gfCNCPoint2[20411] = {X 393.9120, Y 101.1273, Z -3.0000, A 0.000, B 0.000, C 0.000 }
gfCNCPoint2[20412] = {X 393.2786, Y 100.4940, Z -3.0000, A 0.000, B 0.000, C 0.000 }
gfCNCPoint2[20413] = {X 392.8021, Y 99.7355, Z -3.0000, A 0.000, B 0.000, C 0.000 }
gfCNCPoint2[20414] = {X 392.5062, Y 98.8901, Z -3.0000, A 0.000, B 0.000, C 0.000 }
gfCNCPoint2[20415] = {X 392.4059, Y 98.0000, Z -3.0000, A 0.000, B 0.000, C 0.000 }
gfCNCPoint2[20416] = {X 392.4059, Y 97.0659, Z -3.0000, A 0.000, B 0.000, C 0.000 }
gfCNCPoint2[20417] = {X 392.5058, Y 96.1776, Z -3.0000, A 0.000, B 0.000, C 0.000 }
gfCNCPoint2[20418] = {X 392.8005, Y 95.3337, Z -3.0000, A 0.000, B 0.000, C 0.000 }
gfCNCPoint2[20419] = {X 393.2753, Y 94.5762, Z -3.0000, A 0.000, B 0.000, C 0.000 }
gfCNCPoint2[20420] = {X 393.9064, Y 93.9431, Z -3.0000, A 0.000, B 0.000, C 0.000 }
gfCNCPoint2[20421] = {X 394.6623, Y 93.4660, Z -3.0000, A 0.000, B 0.000, C 0.000 }
gfCNCPoint2[20422] = {X 395.5053, Y 93.1686, Z -3.0000, A 0.000, B 0.000, C 0.000 }
gfCNCPoint2[20423] = {X 396.3933, Y 93.0660, Z -3.0000, A 0.000, B 0.000, C 0.000 }
gfCNCPoint2[20424] = {X 397.3648, Y 93.0246, Z -3.0000, A 0.000, B 0.000, C 0.000 }
gfCNCPoint2[20425] = {X 398.3327, Y 92.9326, Z -3.0000, A 0.000, B 0.000, C 0.000 }
gfCNCPoint2[20426] = {X 399.0538, Y 92.7580, Z -3.0000, A 0.000, B 0.000, C 0.000 }
gfCNCPoint2[20427] = {X 399.7177, Y 92.4268, Z -3.0000, A 0.000, B 0.000, C 0.000 }
gfCNCPoint2[20428] = {X 405.3929, Y 88.7698, Z -3.0000, A 0.000, B 0.000, C 0.000 }
gfCNCPoint2[20429] = {X 413.9654, Y 83.2883, Z -3.0000, A 0.000, B 0.000, C 0.000 }
gfCNCPoint2[20430] = {X 411.7675, Y 79.8509, Z -3.0000, A 0.000, B 0.000, C 0.000 }
gfCNCPoint2[20431] = {X 411.7675, Y 79.8509, Z 0.0000, A 0.000, B 0.000, C 0.000 }
gfCNCPoint2[20432] = {X 411.7675, Y 79.8509, Z 11.0000, A 0.000, B 0.000, C 0.000 }
gfCNCPoint2[20433] = {X 466.3102, Y 28.5935, Z 11.0000, A 0.000, B 0.000, C 0.000 }
gfCNCPoint2[20434] = {X 466.3102, Y 28.5935, Z 0.0000, A 0.000, B 0.000, C 0.000 }
gfCNCPoint2[20435] = {X 466.3102, Y 28.5935, Z -3.0000, A 0.000, B 0.000, C 0.000 }
gfCNCPoint2[20436] = {X 462.2302, Y 28.5935, Z -3.0000, A 0.000, B 0.000, C 0.000 }
gfCNCPoint2[20437] = {X 462.2304, Y 40.9130, Z -3.0000, A 0.000, B 0.000, C 0.000 }
gfCNCPoint2[20438] = {X 462.2392, Y 40.9201, Z -3.0000, A 0.000, B 0.000, C 0.000 }
gfCNCPoint2[20439] = {X 462.8741, Y 41.5906, Z -3.0000, A 0.000, B 0.000, C 0.000 }
gfCNCPoint2[20440] = {X 463.3521, Y 42.3808, Z -3.0000, A 0.000, B 0.000, C 0.000 }
gfCNCPoint2[20441] = {X 463.6512, Y 43.2545, Z -3.0000, A 0.000, B 0.000, C 0.000 }
gfCNCPoint2[20442] = {X 463.7578, Y 44.1718, Z -3.0000, A 0.000, B 0.000, C 0.000 }
gfCNCPoint2[20443] = {X 463.7579, Y 45.0000, Z -3.0000, A 0.000, B 0.000, C 0.000 }
gfCNCPoint2[20444] = {X 463.6496, Y 45.9613, Z -3.0000, A 0.000, B 0.000, C 0.000 }
gfCNCPoint2[20445] = {X 463.3301, Y 46.8744, Z -3.0000, A 0.000, B 0.000, C 0.000 }
gfCNCPoint2[20446] = {X 462.8155, Y 47.6935, Z -3.0000, A 0.000, B 0.000, C 0.000 }
gfCNCPoint2[20447] = {X 462.1314, Y 48.3775, Z -3.0000, A 0.000, B 0.000, C 0.000 }
gfCNCPoint2[20448] = {X 461.3123, Y 48.8922, Z -3.0000, A 0.000, B 0.000, C 0.000 }
gfCNCPoint2[20449] = {X 460.3992, Y 49.2117, Z -3.0000, A 0.000, B 0.000, C 0.000 }
gfCNCPoint2[20450] = {X 459.4379, Y 49.3200, Z -3.0000, A 0.000, B 0.000, C 0.000 }
gfCNCPoint2[20451] = {X 452.9945, Y 49.3200, Z -3.0000, A 0.000, B 0.000, C 0.000 }
gfCNCPoint2[20452] = {X 452.0381, Y 49.2128, Z -3.0000, A 0.000, B 0.000, C 0.000 }
gfCNCPoint2[20453] = {X 451.1291, Y 48.8965, Z -3.0000, A 0.000, B 0.000, C 0.000 }
gfCNCPoint2[20454] = {X 450.3127, Y 48.3868, Z -3.0000, A 0.000, B 0.000, C 0.000 }
gfCNCPoint2[20455] = {X 449.6294, Y 47.7091, Z -3.0000, A 0.000, B 0.000, C 0.000 }
gfCNCPoint2[20456] = {X 449.1132, Y 46.8968, Z -3.0000, A 0.000, B 0.000, C 0.000 }
gfCNCPoint2[20457] = {X 448.7895, Y 45.9905, Z -3.0000, A 0.000, B 0.000, C 0.000 }
gfCNCPoint2[20458] = {X 448.6746, Y 45.0349, Z -3.0000, A 0.000, B 0.000, C 0.000 }
gfCNCPoint2[20459] = {X 448.6749, Y 44.1494, Z -3.0000, A 0.000, B 0.000, C 0.000 }
gfCNCPoint2[20460] = {X 448.7853, Y 43.2364, Z -3.0000, A 0.000, B 0.000, C 0.000 }
gfCNCPoint2[20461] = {X 449.0865, Y 42.3675, Z -3.0000, A 0.000, B 0.000, C 0.000 }
gfCNCPoint2[20462] = {X 449.5648, Y 41.5821, Z -3.0000, A 0.000, B 0.000, C 0.000 }
gfCNCPoint2[20463] = {X 450.1984, Y 40.9157, Z -3.0000, A 0.000, B 0.000, C 0.000 }
gfCNCPoint2[20464] = {X 450.1984, Y 34.4738, Z -3.0000, A 0.000, B 0.000, C 0.000 }
gfCNCPoint2[20465] = {X 447.4740, Y 34.4738, Z -3.0000, A 0.000, B 0.000, C 0.000 }
gfCNCPoint2[20466] = {X 443.1893, Y 42.8160, Z -3.0000, A 0.000, B 0.000, C 0.000 }
gfCNCPoint2[20467] = {X 443.1944, Y 42.8296, Z -3.0000, A 0.000, B 0.000, C 0.000 }
gfCNCPoint2[20468] = {X 443.3604, Y 43.4910, Z -3.0000, A 0.000, B 0.000, C 0.000 }
gfCNCPoint2[20469] = {X 443.4203, Y 44.1703, Z -3.0000, A 0.000, B 0.000, C 0.000 }
gfCNCPoint2[20470] = {X 443.4205, Y 45.0000, Z -3.0000, A 0.000, B 0.000, C 0.000 }
gfCNCPoint2[20471] = {X 443.3122, Y 45.9613, Z -3.0000, A 0.000, B 0.000, C 0.000 }
gfCNCPoint2[20472] = {X 442.9927, Y 46.8744, Z -3.0000, A 0.000, B 0.000, C 0.000 }
gfCNCPoint2[20473] = {X 442.4780, Y 47.6935, Z -3.0000, A 0.000, B 0.000, C 0.000 }
gfCNCPoint2[20474] = {X 441.7939, Y 48.3775, Z -3.0000, A 0.000, B 0.000, C 0.000 }
gfCNCPoint2[20475] = {X 440.9748, Y 48.8922, Z -3.0000, A 0.000, B 0.000, C 0.000 }
gfCNCPoint2[20476] = {X 440.0618, Y 49.2117, Z -3.0000, A 0.000, B 0.000, C 0.000 }
gfCNCPoint2[20477] = {X 439.1005, Y 49.3200, Z -3.0000, A 0.000, B 0.000, C 0.000 }
gfCNCPoint2[20478] = {X 432.5144, Y 49.3200, Z -3.0000, A 0.000, B 0.000, C 0.000 }
gfCNCPoint2[20479] = {X 431.5531, Y 49.2117, Z -3.0000, A 0.000, B 0.000, C 0.000 }
gfCNCPoint2[20480] = {X 430.6401, Y 48.8922, Z -3.0000, A 0.000, B 0.000, C 0.000 }
gfCNCPoint2[20481] = {X 429.8210, Y 48.3775, Z -3.0000, A 0.000, B 0.000, C 0.000 }
gfCNCPoint2[20482] = {X 429.1369, Y 47.6935, Z -3.0000, A 0.000, B 0.000, C 0.000 }
gfCNCPoint2[20483] = {X 428.6223, Y 46.8745, Z -3.0000, A 0.000, B 0.000, C 0.000 }
gfCNCPoint2[20484] = {X 428.3027, Y 45.9614, Z -3.0000, A 0.000, B 0.000, C 0.000 }
gfCNCPoint2[20485] = {X 428.1944, Y 45.0001, Z -3.0000, A 0.000, B 0.000, C 0.000 }
gfCNCPoint2[20486] = {X 428.1948, Y 44.1494, Z -3.0000, A 0.000, B 0.000, C 0.000 }
gfCNCPoint2[20487] = {X 428.2925, Y 43.2935, Z -3.0000, A 0.000, B 0.000, C 0.000 }
gfCNCPoint2[20488] = {X 428.5580, Y 42.4740, Z -3.0000, A 0.000, B 0.000, C 0.000 }
gfCNCPoint2[20489] = {X 428.9809, Y 41.7236, Z -3.0000, A 0.000, B 0.000, C 0.000 }
gfCNCPoint2[20490] = {X 429.5442, Y 41.0719, Z -3.0000, A 0.000, B 0.000, C 0.000 }
gfCNCPoint2[20491] = {X 430.2256, Y 40.5449, Z -3.0000, A 0.000, B 0.000, C 0.000 }
gfCNCPoint2[20492] = {X 430.9981, Y 40.1637, Z -3.0000, A 0.000, B 0.000, C 0.000 }
gfCNCPoint2[20493] = {X 434.9873, Y 32.3552, Z -3.0000, A 0.000, B 0.000, C 0.000 }
gfCNCPoint2[20494] = {X 433.8174, Y 31.5687, Z -3.0000, A 0.000, B 0.000, C 0.000 }
gfCNCPoint2[20495] = {X 432.7544, Y 30.6429, Z -3.0000, A 0.000, B 0.000, C 0.000 }
gfCNCPoint2[20496] = {X 431.8146, Y 29.5922, Z -3.0000, A 0.000, B 0.000, C 0.000 }
gfCNCPoint2[20497] = {X 431.0127, Y 28.4328, Z -3.0000, A 0.000, B 0.000, C 0.000 }
gfCNCPoint2[20498] = {X 430.3611, Y 27.1828, Z -3.0000, A 0.000, B 0.000, C 0.000 }
gfCNCPoint2[20499] = {X 429.8699, Y 25.8615, Z -3.0000, A 0.000, B 0.000, C 0.000 }
gfCNCPoint2[20500] = {X 429.4508, Y 24.0500, Z -3.0000, A 0.000, B 0.000, C 0.000 }
gfCNCPoint2[20501] = {X 429.2372, Y 22.2029, Z -3.0000, A 0.000, B 0.000, C 0.000 }
gfCNCPoint2[20502] = {X 429.2318, Y 20.3436, Z -3.0000, A 0.000, B 0.000, C 0.000 }
gfCNCPoint2[20503] = {X 429.4347, Y 18.4953, Z -3.0000, A 0.000, B 0.000, C 0.000 }
gfCNCPoint2[20504] = {X 429.8434, Y 16.6814, Z -3.0000, A 0.000, B 0.000, C 0.000 }
gfCNCPoint2[20505] = {X 430.3648, Y 15.2116, Z -3.0000, A 0.000, B 0.000, C 0.000 }
gfCNCPoint2[20506] = {X 431.0757, Y 13.8235, Z -3.0000, A 0.000, B 0.000, C 0.000 }
gfCNCPoint2[20507] = {X 431.9635, Y 12.5413, Z -3.0000, A 0.000, B 0.000, C 0.000 }
gfCNCPoint2[20508] = {X 433.0127, Y 11.3874, Z -3.0000, A 0.000, B 0.000, C 0.000 }
gfCNCPoint2[20509] = {X 434.2050, Y 10.3821, Z -3.0000, A 0.000, B 0.000, C 0.000 }
gfCNCPoint2[20510] = {X 435.5195, Y 9.5429, Z -3.0000, A 0.000, B 0.000, C 0.000 }
gfCNCPoint2[20511] = {X 436.9333, Y 8.8845, Z -3.0000, A 0.000, B 0.000, C 0.000 }
gfCNCPoint2[20512] = {X 438.4216, Y 8.4184, Z -3.0000, A 0.000, B 0.000, C 0.000 }
gfCNCPoint2[20513] = {X 440.0467, Y 8.1096, Z -3.0000, A 0.000, B 0.000, C 0.000 }
gfCNCPoint2[20514] = {X 441.6910, Y 7.9282, Z -3.0000, A 0.000, B 0.000, C 0.000 }
gfCNCPoint2[20515] = {X 443.3444, Y 7.8753, Z -3.0000, A 0.000, B 0.000, C 0.000 }
gfCNCPoint2[20516] = {X 444.0357, Y 7.8712, Z -3.0000, A 0.000, B 0.000, C 0.000 }
gfCNCPoint2[20517] = {X 459.4466, Y 7.8712, Z -3.0000, A 0.000, B 0.000, C 0.000 }
gfCNCPoint2[20518] = {X 460.4060, Y 7.9793, Z -3.0000, A 0.000, B 0.000, C 0.000 }
gfCNCPoint2[20519] = {X 461.3172, Y 8.2982, Z -3.0000, A 0.000, B 0.000, C 0.000 }
gfCNCPoint2[20520] = {X 462.1347, Y 8.8118, Z -3.0000, A 0.000, B 0.000, C 0.000 }
gfCNCPoint2[20521] = {X 462.8173, Y 9.4945, Z -3.0000, A 0.000, B 0.000, C 0.000 }
gfCNCPoint2[20522] = {X 463.3310, Y 10.3120, Z -3.0000, A 0.000, B 0.000, C 0.000 }
gfCNCPoint2[20523] = {X 463.6498, Y 11.2232, Z -3.0000, A 0.000, B 0.000, C 0.000 }
gfCNCPoint2[20524] = {X 463.7579, Y 12.1826, Z -3.0000, A 0.000, B 0.000, C 0.000 }
gfCNCPoint2[20525] = {X 463.7579, Y 12.9781, Z -3.0000, A 0.000, B 0.000, C 0.000 }
gfCNCPoint2[20526] = {X 463.6565, Y 13.9081, Z -3.0000, A 0.000, B 0.000, C 0.000 }
gfCNCPoint2[20527] = {X 463.3573, Y 14.7945, Z -3.0000, A 0.000, B 0.000, C 0.000 }
gfCNCPoint2[20528] = {X 462.8742, Y 15.5957, Z -3.0000, A 0.000, B 0.000, C 0.000 }
gfCNCPoint2[20529] = {X 462.2300, Y 16.2741, Z -3.0000, A 0.000, B 0.000, C 0.000 }
gfCNCPoint2[20530] = {X 462.2302, Y 28.5935, Z -3.0000, A 0.000, B 0.000, C 0.000 }
gfCNCPoint2[20531] = {X 466.2302, Y 28.5935, Z -3.0000, A 0.000, B 0.000, C 0.000 }
gfCNCPoint2[20532] = {X 462.1502, Y 28.5935, Z -3.0000, A 0.000, B 0.000, C 0.000 }
gfCNCPoint2[20533] = {X 462.1504, Y 40.9512, Z -3.0000, A 0.000, B 0.000, C 0.000 }
gfCNCPoint2[20534] = {X 462.1880, Y 40.9816, Z -3.0000, A 0.000, B 0.000, C 0.000 }
gfCNCPoint2[20535] = {X 462.8110, Y 41.6397, Z -3.0000, A 0.000, B 0.000, C 0.000 }
gfCNCPoint2[20536] = {X 463.2798, Y 42.4151, Z -3.0000, A 0.000, B 0.000, C 0.000 }
gfCNCPoint2[20537] = {X 463.5732, Y 43.2724, Z -3.0000, A 0.000, B 0.000, C 0.000 }
gfCNCPoint2[20538] = {X 463.6778, Y 44.1724, Z -3.0000, A 0.000, B 0.000, C 0.000 }
gfCNCPoint2[20539] = {X 463.6779, Y 45.0000, Z -3.0000, A 0.000, B 0.000, C 0.000 }
gfCNCPoint2[20540] = {X 463.5716, Y 45.9435, Z -3.0000, A 0.000, B 0.000, C 0.000 }
gfCNCPoint2[20541] = {X 463.2580, Y 46.8397, Z -3.0000, A 0.000, B 0.000, C 0.000 }
gfCNCPoint2[20542] = {X 462.7529, Y 47.6436, Z -3.0000, A 0.000, B 0.000, C 0.000 }
gfCNCPoint2[20543] = {X 462.0815, Y 48.3150, Z -3.0000, A 0.000, B 0.000, C 0.000 }
gfCNCPoint2[20544] = {X 461.2776, Y 48.8201, Z -3.0000, A 0.000, B 0.000, C 0.000 }
gfCNCPoint2[20545] = {X 460.3814, Y 49.1337, Z -3.0000, A 0.000, B 0.000, C 0.000 }
gfCNCPoint2[20546] = {X 459.4379, Y 49.2400, Z -3.0000, A 0.000, B 0.000, C 0.000 }
gfCNCPoint2[20547] = {X 452.9945, Y 49.2400, Z -3.0000, A 0.000, B 0.000, C 0.000 }
gfCNCPoint2[20548] = {X 452.0558, Y 49.1348, Z -3.0000, A 0.000, B 0.000, C 0.000 }
gfCNCPoint2[20549] = {X 451.1636, Y 48.8243, Z -3.0000, A 0.000, B 0.000, C 0.000 }
gfCNCPoint2[20550] = {X 450.3624, Y 48.3241, Z -3.0000, A 0.000, B 0.000, C 0.000 }
gfCNCPoint2[20551] = {X 449.6918, Y 47.6589, Z -3.0000, A 0.000, B 0.000, C 0.000 }
gfCNCPoint2[20552] = {X 449.1851, Y 46.8617, Z -3.0000, A 0.000, B 0.000, C 0.000 }
gfCNCPoint2[20553] = {X 448.8674, Y 45.9721, Z -3.0000, A 0.000, B 0.000, C 0.000 }
gfCNCPoint2[20554] = {X 448.7546, Y 45.0343, Z -3.0000, A 0.000, B 0.000, C 0.000 }
gfCNCPoint2[20555] = {X 448.7549, Y 44.1505, Z -3.0000, A 0.000, B 0.000, C 0.000 }
gfCNCPoint2[20556] = {X 448.8654, Y 43.2454, Z -3.0000, A 0.000, B 0.000, C 0.000 }
gfCNCPoint2[20557] = {X 449.1668, Y 42.3850, Z -3.0000, A 0.000, B 0.000, C 0.000 }
gfCNCPoint2[20558] = {X 449.6452, Y 41.6088, Z -3.0000, A 0.000, B 0.000, C 0.000 }
gfCNCPoint2[20559] = {X 450.2784, Y 40.9529, Z -3.0000, A 0.000, B 0.000, C 0.000 }
gfCNCPoint2[20560] = {X 450.2784, Y 34.3938, Z -3.0000, A 0.000, B 0.000, C 0.000 }
gfCNCPoint2[20561] = {X 447.4251, Y 34.3938, Z -3.0000, A 0.000, B 0.000, C 0.000 }
gfCNCPoint2[20562] = {X 443.1021, Y 42.8107, Z -3.0000, A 0.000, B 0.000, C 0.000 }
gfCNCPoint2[20563] = {X 443.1190, Y 42.8563, Z -3.0000, A 0.000, B 0.000, C 0.000 }
gfCNCPoint2[20564] = {X 443.2816, Y 43.5049, Z -3.0000, A 0.000, B 0.000, C 0.000 }
gfCNCPoint2[20565] = {X 443.3403, Y 44.1710, Z -3.0000, A 0.000, B 0.000, C 0.000 }
gfCNCPoint2[20566] = {X 443.3405, Y 45.0000, Z -3.0000, A 0.000, B 0.000, C 0.000 }
gfCNCPoint2[20567] = {X 443.2342, Y 45.9435, Z -3.0000, A 0.000, B 0.000, C 0.000 }
gfCNCPoint2[20568] = {X 442.9206, Y 46.8397, Z -3.0000, A 0.000, B 0.000, C 0.000 }
gfCNCPoint2[20569] = {X 442.4154, Y 47.6436, Z -3.0000, A 0.000, B 0.000, C 0.000 }
gfCNCPoint2[20570] = {X 441.7441, Y 48.3150, Z -3.0000, A 0.000, B 0.000, C 0.000 }
gfCNCPoint2[20571] = {X 440.9401, Y 48.8201, Z -3.0000, A 0.000, B 0.000, C 0.000 }
gfCNCPoint2[20572] = {X 440.0440, Y 49.1337, Z -3.0000, A 0.000, B 0.000, C 0.000 }
gfCNCPoint2[20573] = {X 439.1005, Y 49.2400, Z -3.0000, A 0.000, B 0.000, C 0.000 }
gfCNCPoint2[20574] = {X 432.5144, Y 49.2400, Z -3.0000, A 0.000, B 0.000, C 0.000 }
gfCNCPoint2[20575] = {X 431.5709, Y 49.1337, Z -3.0000, A 0.000, B 0.000, C 0.000 }
gfCNCPoint2[20576] = {X 430.6748, Y 48.8201, Z -3.0000, A 0.000, B 0.000, C 0.000 }
gfCNCPoint2[20577] = {X 429.8708, Y 48.3150, Z -3.0000, A 0.000, B 0.000, C 0.000 }
gfCNCPoint2[20578] = {X 429.1995, Y 47.6436, Z -3.0000, A 0.000, B 0.000, C 0.000 }
gfCNCPoint2[20579] = {X 428.6943, Y 46.8397, Z -3.0000, A 0.000, B 0.000, C 0.000 }
gfCNCPoint2[20580] = {X 428.3807, Y 45.9436, Z -3.0000, A 0.000, B 0.000, C 0.000 }
gfCNCPoint2[20581] = {X 428.2744, Y 45.0001, Z -3.0000, A 0.000, B 0.000, C 0.000 }
gfCNCPoint2[20582] = {X 428.2748, Y 44.1505, Z -3.0000, A 0.000, B 0.000, C 0.000 }
gfCNCPoint2[20583] = {X 428.3718, Y 43.3054, Z -3.0000, A 0.000, B 0.000, C 0.000 }
gfCNCPoint2[20584] = {X 428.6354, Y 42.4967, Z -3.0000, A 0.000, B 0.000, C 0.000 }
gfCNCPoint2[20585] = {X 429.0552, Y 41.7570, Z -3.0000, A 0.000, B 0.000, C 0.000 }
gfCNCPoint2[20586] = {X 429.6142, Y 41.1159, Z -3.0000, A 0.000, B 0.000, C 0.000 }
gfCNCPoint2[20587] = {X 430.2899, Y 40.5992, Z -3.0000, A 0.000, B 0.000, C 0.000 }
gfCNCPoint2[20588] = {X 431.0551, Y 40.2278, Z -3.0000, A 0.000, B 0.000, C 0.000 }
gfCNCPoint2[20589] = {X 435.0930, Y 32.3241, Z -3.0000, A 0.000, B 0.000, C 0.000 }
gfCNCPoint2[20590] = {X 433.9162, Y 31.5434, Z -3.0000, A 0.000, B 0.000, C 0.000 }
gfCNCPoint2[20591] = {X 432.8465, Y 30.6212, Z -3.0000, A 0.000, B 0.000, C 0.000 }
gfCNCPoint2[20592] = {X 431.9009, Y 29.5723, Z -3.0000, A 0.000, B 0.000, C 0.000 }
gfCNCPoint2[20593] = {X 431.0943, Y 28.4130, Z -3.0000, A 0.000, B 0.000, C 0.000 }
gfCNCPoint2[20594] = {X 430.4394, Y 27.1618, Z -3.0000, A 0.000, B 0.000, C 0.000 }
gfCNCPoint2[20595] = {X 429.9465, Y 25.8383, Z -3.0000, A 0.000, B 0.000, C 0.000 }
gfCNCPoint2[20596] = {X 429.5295, Y 24.0357, Z -3.0000, A 0.000, B 0.000, C 0.000 }
gfCNCPoint2[20597] = {X 429.3171, Y 22.1977, Z -3.0000, A 0.000, B 0.000, C 0.000 }
gfCNCPoint2[20598] = {X 429.3117, Y 20.3474, Z -3.0000, A 0.000, B 0.000, C 0.000 }
gfCNCPoint2[20599] = {X 429.5137, Y 18.5082, Z -3.0000, A 0.000, B 0.000, C 0.000 }
gfCNCPoint2[20600] = {X 429.9203, Y 16.7032, Z -3.0000, A 0.000, B 0.000, C 0.000 }
gfCNCPoint2[20601] = {X 430.4383, Y 15.2434, Z -3.0000, A 0.000, B 0.000, C 0.000 }
gfCNCPoint2[20602] = {X 431.1443, Y 13.8646, Z -3.0000, A 0.000, B 0.000, C 0.000 }
gfCNCPoint2[20603] = {X 432.0261, Y 12.5911, Z -3.0000, A 0.000, B 0.000, C 0.000 }
gfCNCPoint2[20604] = {X 433.0682, Y 11.4451, Z -3.0000, A 0.000, B 0.000, C 0.000 }
gfCNCPoint2[20605] = {X 434.2524, Y 10.4466, Z -3.0000, A 0.000, B 0.000, C 0.000 }
gfCNCPoint2[20606] = {X 435.5580, Y 9.6131, Z -3.0000, A 0.000, B 0.000, C 0.000 }
gfCNCPoint2[20607] = {X 436.9622, Y 8.9591, Z -3.0000, A 0.000, B 0.000, C 0.000 }
gfCNCPoint2[20608] = {X 438.4404, Y 8.4961, Z -3.0000, A 0.000, B 0.000, C 0.000 }
gfCNCPoint2[20609] = {X 440.0593, Y 8.1886, Z -3.0000, A 0.000, B 0.000, C 0.000 }
gfCNCPoint2[20610] = {X 441.6973, Y 8.0079, Z -3.0000, A 0.000, B 0.000, C 0.000 }
gfCNCPoint2[20611] = {X 443.3443, Y 7.9553, Z -3.0000, A 0.000, B 0.000, C 0.000 }
gfCNCPoint2[20612] = {X 444.0360, Y 7.9512, Z -3.0000, A 0.000, B 0.000, C 0.000 }
gfCNCPoint2[20613] = {X 459.4466, Y 7.9512, Z -3.0000, A 0.000, B 0.000, C 0.000 }
gfCNCPoint2[20614] = {X 460.3882, Y 8.0573, Z -3.0000, A 0.000, B 0.000, C 0.000 }
gfCNCPoint2[20615] = {X 461.2825, Y 8.3703, Z -3.0000, A 0.000, B 0.000, C 0.000 }
gfCNCPoint2[20616] = {X 462.0848, Y 8.8744, Z -3.0000, A 0.000, B 0.000, C 0.000 }
gfCNCPoint2[20617] = {X 462.7548, Y 9.5444, Z -3.0000, A 0.000, B 0.000, C 0.000 }
gfCNCPoint2[20618] = {X 463.2589, Y 10.3467, Z -3.0000, A 0.000, B 0.000, C 0.000 }
gfCNCPoint2[20619] = {X 463.5719, Y 11.2410, Z -3.0000, A 0.000, B 0.000, C 0.000 }
gfCNCPoint2[20620] = {X 463.6779, Y 12.1826, Z -3.0000, A 0.000, B 0.000, C 0.000 }
gfCNCPoint2[20621] = {X 463.6779, Y 12.9781, Z -3.0000, A 0.000, B 0.000, C 0.000 }
gfCNCPoint2[20622] = {X 463.5764, Y 13.8999, Z -3.0000, A 0.000, B 0.000, C 0.000 }
gfCNCPoint2[20623] = {X 463.2769, Y 14.7776, Z -3.0000, A 0.000, B 0.000, C 0.000 }
gfCNCPoint2[20624] = {X 462.7937, Y 15.5692, Z -3.0000, A 0.000, B 0.000, C 0.000 }
gfCNCPoint2[20625] = {X 462.1500, Y 16.2368, Z -3.0000, A 0.000, B 0.000, C 0.000 }
gfCNCPoint2[20626] = {X 462.1502, Y 28.5935, Z -3.0000, A 0.000, B 0.000, C 0.000 }
gfCNCPoint2[20627] = {X 466.1502, Y 28.5935, Z -3.0000, A 0.000, B 0.000, C 0.000 }
gfCNCPoint2[20628] = {X 462.0702, Y 28.5935, Z -3.0000, A 0.000, B 0.000, C 0.000 }
gfCNCPoint2[20629] = {X 462.0704, Y 40.9893, Z -3.0000, A 0.000, B 0.000, C 0.000 }
gfCNCPoint2[20630] = {X 462.1369, Y 41.0431, Z -3.0000, A 0.000, B 0.000, C 0.000 }
gfCNCPoint2[20631] = {X 462.7478, Y 41.6887, Z -3.0000, A 0.000, B 0.000, C 0.000 }
gfCNCPoint2[20632] = {X 463.2075, Y 42.4493, Z -3.0000, A 0.000, B 0.000, C 0.000 }
gfCNCPoint2[20633] = {X 463.4953, Y 43.2903, Z -3.0000, A 0.000, B 0.000, C 0.000 }
gfCNCPoint2[20634] = {X 463.5978, Y 44.1731, Z -3.0000, A 0.000, B 0.000, C 0.000 }
gfCNCPoint2[20635] = {X 463.5979, Y 45.0000, Z -3.0000, A 0.000, B 0.000, C 0.000 }
gfCNCPoint2[20636] = {X 463.4936, Y 45.9257, Z -3.0000, A 0.000, B 0.000, C 0.000 }
gfCNCPoint2[20637] = {X 463.1860, Y 46.8050, Z -3.0000, A 0.000, B 0.000, C 0.000 }
gfCNCPoint2[20638] = {X 462.6904, Y 47.5937, Z -3.0000, A 0.000, B 0.000, C 0.000 }
gfCNCPoint2[20639] = {X 462.0317, Y 48.2524, Z -3.0000, A 0.000, B 0.000, C 0.000 }
gfCNCPoint2[20640] = {X 461.2429, Y 48.7480, Z -3.0000, A 0.000, B 0.000, C 0.000 }
gfCNCPoint2[20641] = {X 460.3636, Y 49.0557, Z -3.0000, A 0.000, B 0.000, C 0.000 }
gfCNCPoint2[20642] = {X 459.4379, Y 49.1600, Z -3.0000, A 0.000, B 0.000, C 0.000 }
gfCNCPoint2[20643] = {X 452.9945, Y 49.1600, Z -3.0000, A 0.000, B 0.000, C 0.000 }
gfCNCPoint2[20644] = {X 452.0735, Y 49.0568, Z -3.0000, A 0.000, B 0.000, C 0.000 }
gfCNCPoint2[20645] = {X 451.1982, Y 48.7522, Z -3.0000, A 0.000, B 0.000, C 0.000 }
gfCNCPoint2[20646] = {X 450.4120, Y 48.2614, Z -3.0000, A 0.000, B 0.000, C 0.000 }
gfCNCPoint2[20647] = {X 449.7541, Y 47.6087, Z -3.0000, A 0.000, B 0.000, C 0.000 }
gfCNCPoint2[20648] = {X 449.2569, Y 46.8266, Z -3.0000, A 0.000, B 0.000, C 0.000 }
gfCNCPoint2[20649] = {X 448.9453, Y 45.9538, Z -3.0000, A 0.000, B 0.000, C 0.000 }
gfCNCPoint2[20650] = {X 448.8346, Y 45.0336, Z -3.0000, A 0.000, B 0.000, C 0.000 }
gfCNCPoint2[20651] = {X 448.8349, Y 44.1516, Z -3.0000, A 0.000, B 0.000, C 0.000 }
gfCNCPoint2[20652] = {X 448.9454, Y 43.2545, Z -3.0000, A 0.000, B 0.000, C 0.000 }
gfCNCPoint2[20653] = {X 449.2471, Y 42.4026, Z -3.0000, A 0.000, B 0.000, C 0.000 }
gfCNCPoint2[20654] = {X 449.7256, Y 41.6358, Z -3.0000, A 0.000, B 0.000, C 0.000 }
gfCNCPoint2[20655] = {X 450.3584, Y 40.9906, Z -3.0000, A 0.000, B 0.000, C 0.000 }
gfCNCPoint2[20656] = {X 450.3584, Y 34.3138, Z -3.0000, A 0.000, B 0.000, C 0.000 }
gfCNCPoint2[20657] = {X 447.3763, Y 34.3138, Z -3.0000, A 0.000, B 0.000, C 0.000 }
gfCNCPoint2[20658] = {X 443.0148, Y 42.8055, Z -3.0000, A 0.000, B 0.000, C 0.000 }
gfCNCPoint2[20659] = {X 443.0435, Y 42.8830, Z -3.0000, A 0.000, B 0.000, C 0.000 }
gfCNCPoint2[20660] = {X 443.2028, Y 43.5188, Z -3.0000, A 0.000, B 0.000, C 0.000 }
gfCNCPoint2[20661] = {X 443.2603, Y 44.1717, Z -3.0000, A 0.000, B 0.000, C 0.000 }
gfCNCPoint2[20662] = {X 443.2605, Y 45.0000, Z -3.0000, A 0.000, B 0.000, C 0.000 }
gfCNCPoint2[20663] = {X 443.1562, Y 45.9257, Z -3.0000, A 0.000, B 0.000, C 0.000 }
gfCNCPoint2[20664] = {X 442.8485, Y 46.8050, Z -3.0000, A 0.000, B 0.000, C 0.000 }
gfCNCPoint2[20665] = {X 442.3529, Y 47.5937, Z -3.0000, A 0.000, B 0.000, C 0.000 }
gfCNCPoint2[20666] = {X 441.6942, Y 48.2524, Z -3.0000, A 0.000, B 0.000, C 0.000 }
gfCNCPoint2[20667] = {X 440.9054, Y 48.7480, Z -3.0000, A 0.000, B 0.000, C 0.000 }
gfCNCPoint2[20668] = {X 440.0262, Y 49.0557, Z -3.0000, A 0.000, B 0.000, C 0.000 }
gfCNCPoint2[20669] = {X 439.1005, Y 49.1600, Z -3.0000, A 0.000, B 0.000, C 0.000 }
gfCNCPoint2[20670] = {X 432.5144, Y 49.1600, Z -3.0000, A 0.000, B 0.000, C 0.000 }
gfCNCPoint2[20671] = {X 431.5887, Y 49.0557, Z -3.0000, A 0.000, B 0.000, C 0.000 }
gfCNCPoint2[20672] = {X 430.7095, Y 48.7480, Z -3.0000, A 0.000, B 0.000, C 0.000 }
gfCNCPoint2[20673] = {X 429.9207, Y 48.2524, Z -3.0000, A 0.000, B 0.000, C 0.000 }
gfCNCPoint2[20674] = {X 429.2620, Y 47.5937, Z -3.0000, A 0.000, B 0.000, C 0.000 }
gfCNCPoint2[20675] = {X 428.7664, Y 46.8050, Z -3.0000, A 0.000, B 0.000, C 0.000 }
gfCNCPoint2[20676] = {X 428.4587, Y 45.9257, Z -3.0000, A 0.000, B 0.000, C 0.000 }
gfCNCPoint2[20677] = {X 428.3544, Y 45.0000, Z -3.0000, A 0.000, B 0.000, C 0.000 }
gfCNCPoint2[20678] = {X 428.3548, Y 44.1516, Z -3.0000, A 0.000, B 0.000, C 0.000 }
gfCNCPoint2[20679] = {X 428.4510, Y 43.3174, Z -3.0000, A 0.000, B 0.000, C 0.000 }
gfCNCPoint2[20680] = {X 428.7128, Y 42.5195, Z -3.0000, A 0.000, B 0.000, C 0.000 }
gfCNCPoint2[20681] = {X 429.1295, Y 41.7905, Z -3.0000, A 0.000, B 0.000, C 0.000 }
gfCNCPoint2[20682] = {X 429.6841, Y 41.1600, Z -3.0000, A 0.000, B 0.000, C 0.000 }
gfCNCPoint2[20683] = {X 430.3541, Y 40.6537, Z -3.0000, A 0.000, B 0.000, C 0.000 }
gfCNCPoint2[20684] = {X 431.1120, Y 40.2923, Z -3.0000, A 0.000, B 0.000, C 0.000 }
gfCNCPoint2[20685] = {X 435.1990, Y 32.2925, Z -3.0000, A 0.000, B 0.000, C 0.000 }
gfCNCPoint2[20686] = {X 434.0151, Y 31.5177, Z -3.0000, A 0.000, B 0.000, C 0.000 }
gfCNCPoint2[20687] = {X 432.9388, Y 30.5994, Z -3.0000, A 0.000, B 0.000, C 0.000 }
gfCNCPoint2[20688] = {X 431.9872, Y 29.5523, Z -3.0000, A 0.000, B 0.000, C 0.000 }
gfCNCPoint2[20689] = {X 431.1758, Y 28.3932, Z -3.0000, A 0.000, B 0.000, C 0.000 }
gfCNCPoint2[20690] = {X 430.5176, Y 27.1408, Z -3.0000, A 0.000, B 0.000, C 0.000 }
gfCNCPoint2[20691] = {X 430.0231, Y 25.8152, Z -3.0000, A 0.000, B 0.000, C 0.000 }
gfCNCPoint2[20692] = {X 429.6082, Y 24.0214, Z -3.0000, A 0.000, B 0.000, C 0.000 }
gfCNCPoint2[20693] = {X 429.3969, Y 22.1924, Z -3.0000, A 0.000, B 0.000, C 0.000 }
gfCNCPoint2[20694] = {X 429.3917, Y 20.3513, Z -3.0000, A 0.000, B 0.000, C 0.000 }
gfCNCPoint2[20695] = {X 429.5926, Y 18.5212, Z -3.0000, A 0.000, B 0.000, C 0.000 }
gfCNCPoint2[20696] = {X 429.9973, Y 16.7250, Z -3.0000, A 0.000, B 0.000, C 0.000 }
gfCNCPoint2[20697] = {X 430.5117, Y 15.2752, Z -3.0000, A 0.000, B 0.000, C 0.000 }
gfCNCPoint2[20698] = {X 431.2129, Y 13.9058, Z -3.0000, A 0.000, B 0.000, C 0.000 }
gfCNCPoint2[20699] = {X 432.0886, Y 12.6410, Z -3.0000, A 0.000, B 0.000, C 0.000 }
gfCNCPoint2[20700] = {X 433.1236, Y 11.5027, Z -3.0000, A 0.000, B 0.000, C 0.000 }
gfCNCPoint2[20701] = {X 434.2998, Y 10.5110, Z -3.0000, A 0.000, B 0.000, C 0.000 }
gfCNCPoint2[20702] = {X 435.5965, Y 9.6832, Z -3.0000, A 0.000, B 0.000, C 0.000 }
gfCNCPoint2[20703] = {X 436.9911, Y 9.0337, Z -3.0000, A 0.000, B 0.000, C 0.000 }
gfCNCPoint2[20704] = {X 438.4592, Y 8.5739, Z -3.0000, A 0.000, B 0.000, C 0.000 }
gfCNCPoint2[20705] = {X 440.0719, Y 8.2676, Z -3.0000, A 0.000, B 0.000, C 0.000 }
gfCNCPoint2[20706] = {X 441.7036, Y 8.0877, Z -3.0000, A 0.000, B 0.000, C 0.000 }
gfCNCPoint2[20707] = {X 443.3443, Y 8.0353, Z -3.0000, A 0.000, B 0.000, C 0.000 }
gfCNCPoint2[20708] = {X 444.0362, Y 8.0312, Z -3.0000, A 0.000, B 0.000, C 0.000 }
gfCNCPoint2[20709] = {X 459.4466, Y 8.0312, Z -3.0000, A 0.000, B 0.000, C 0.000 }
gfCNCPoint2[20710] = {X 460.3703, Y 8.1353, Z -3.0000, A 0.000, B 0.000, C 0.000 }
gfCNCPoint2[20711] = {X 461.2478, Y 8.4423, Z -3.0000, A 0.000, B 0.000, C 0.000 }
gfCNCPoint2[20712] = {X 462.0349, Y 8.9369, Z -3.0000, A 0.000, B 0.000, C 0.000 }
gfCNCPoint2[20713] = {X 462.6922, Y 9.5943, Z -3.0000, A 0.000, B 0.000, C 0.000 }
gfCNCPoint2[20714] = {X 463.1868, Y 10.3814, Z -3.0000, A 0.000, B 0.000, C 0.000 }
gfCNCPoint2[20715] = {X 463.4939, Y 11.2588, Z -3.0000, A 0.000, B 0.000, C 0.000 }
gfCNCPoint2[20716] = {X 463.5979, Y 12.1826, Z -3.0000, A 0.000, B 0.000, C 0.000 }
gfCNCPoint2[20717] = {X 463.5979, Y 12.9781, Z -3.0000, A 0.000, B 0.000, C 0.000 }
gfCNCPoint2[20718] = {X 463.5022, Y 13.8653, Z -3.0000, A 0.000, B 0.000, C 0.000 }
gfCNCPoint2[20719] = {X 463.2195, Y 14.7116, Z -3.0000, A 0.000, B 0.000, C 0.000 }
gfCNCPoint2[20720] = {X 462.7629, Y 15.4781, Z -3.0000, A 0.000, B 0.000, C 0.000 }
gfCNCPoint2[20721] = {X 462.1532, Y 16.1297, Z -3.0000, A 0.000, B 0.000, C 0.000 }
gfCNCPoint2[20722] = {X 462.0700, Y 16.1995, Z -3.0000, A 0.000, B 0.000, C 0.000 }
gfCNCPoint2[20723] = {X 462.0702, Y 28.5935, Z -3.0000, A 0.000, B 0.000, C 0.000 }
gfCNCPoint2[20724] = {X 466.0702, Y 28.5935, Z -3.0000, A 0.000, B 0.000, C 0.000 }
gfCNCPoint2[20725] = {X 461.9902, Y 28.5935, Z -3.0000, A 0.000, B 0.000, C 0.000 }
gfCNCPoint2[20726] = {X 461.9904, Y 41.0275, Z -3.0000, A 0.000, B 0.000, C 0.000 }
gfCNCPoint2[20727] = {X 462.0857, Y 41.1047, Z -3.0000, A 0.000, B 0.000, C 0.000 }
gfCNCPoint2[20728] = {X 462.6846, Y 41.7378, Z -3.0000, A 0.000, B 0.000, C 0.000 }
gfCNCPoint2[20729] = {X 463.1353, Y 42.4836, Z -3.0000, A 0.000, B 0.000, C 0.000 }
gfCNCPoint2[20730] = {X 463.4173, Y 43.3082, Z -3.0000, A 0.000, B 0.000, C 0.000 }
gfCNCPoint2[20731] = {X 463.5178, Y 44.1738, Z -3.0000, A 0.000, B 0.000, C 0.000 }
gfCNCPoint2[20732] = {X 463.5179, Y 45.0000, Z -3.0000, A 0.000, B 0.000, C 0.000 }
gfCNCPoint2[20733] = {X 463.4156, Y 45.9079, Z -3.0000, A 0.000, B 0.000, C 0.000 }
gfCNCPoint2[20734] = {X 463.1139, Y 46.7702, Z -3.0000, A 0.000, B 0.000, C 0.000 }
gfCNCPoint2[20735] = {X 462.6278, Y 47.5438, Z -3.0000, A 0.000, B 0.000, C 0.000 }
gfCNCPoint2[20736] = {X 461.9818, Y 48.1899, Z -3.0000, A 0.000, B 0.000, C 0.000 }
gfCNCPoint2[20737] = {X 461.2082, Y 48.6760, Z -3.0000, A 0.000, B 0.000, C 0.000 }
gfCNCPoint2[20738] = {X 460.3458, Y 48.9777, Z -3.0000, A 0.000, B 0.000, C 0.000 }
gfCNCPoint2[20739] = {X 459.4379, Y 49.0800, Z -3.0000, A 0.000, B 0.000, C 0.000 }
gfCNCPoint2[20740] = {X 452.9945, Y 49.0800, Z -3.0000, A 0.000, B 0.000, C 0.000 }
gfCNCPoint2[20741] = {X 452.0912, Y 48.9788, Z -3.0000, A 0.000, B 0.000, C 0.000 }
gfCNCPoint2[20742] = {X 451.2327, Y 48.6800, Z -3.0000, A 0.000, B 0.000, C 0.000 }
gfCNCPoint2[20743] = {X 450.4617, Y 48.1987, Z -3.0000, A 0.000, B 0.000, C 0.000 }
gfCNCPoint2[20744] = {X 449.8164, Y 47.5585, Z -3.0000, A 0.000, B 0.000, C 0.000 }
gfCNCPoint2[20745] = {X 449.3288, Y 46.7914, Z -3.0000, A 0.000, B 0.000, C 0.000 }
gfCNCPoint2[20746] = {X 449.0232, Y 45.9354, Z -3.0000, A 0.000, B 0.000, C 0.000 }
gfCNCPoint2[20747] = {X 448.9146, Y 45.0330, Z -3.0000, A 0.000, B 0.000, C 0.000 }
gfCNCPoint2[20748] = {X 448.9149, Y 44.1527, Z -3.0000, A 0.000, B 0.000, C 0.000 }
gfCNCPoint2[20749] = {X 449.0254, Y 43.2637, Z -3.0000, A 0.000, B 0.000, C 0.000 }
gfCNCPoint2[20750] = {X 449.3274, Y 42.4203, Z -3.0000, A 0.000, B 0.000, C 0.000 }
gfCNCPoint2[20751] = {X 449.8061, Y 41.6631, Z -3.0000, A 0.000, B 0.000, C 0.000 }
gfCNCPoint2[20752] = {X 450.4384, Y 41.0287, Z -3.0000, A 0.000, B 0.000, C 0.000 }
gfCNCPoint2[20753] = {X 450.4384, Y 34.2338, Z -3.0000, A 0.000, B 0.000, C 0.000 }
gfCNCPoint2[20754] = {X 447.3275, Y 34.2338, Z -3.0000, A 0.000, B 0.000, C 0.000 }
gfCNCPoint2[20755] = {X 442.9276, Y 42.8003, Z -3.0000, A 0.000, B 0.000, C 0.000 }
gfCNCPoint2[20756] = {X 442.9681, Y 42.9096, Z -3.0000, A 0.000, B 0.000, C 0.000 }
gfCNCPoint2[20757] = {X 443.1241, Y 43.5327, Z -3.0000, A 0.000, B 0.000, C 0.000 }
gfCNCPoint2[20758] = {X 443.1803, Y 44.1725, Z -3.0000, A 0.000, B 0.000, C 0.000 }
gfCNCPoint2[20759] = {X 443.1805, Y 45.0000, Z -3.0000, A 0.000, B 0.000, C 0.000 }
gfCNCPoint2[20760] = {X 443.0782, Y 45.9079, Z -3.0000, A 0.000, B 0.000, C 0.000 }
gfCNCPoint2[20761] = {X 442.7764, Y 46.7702, Z -3.0000, A 0.000, B 0.000, C 0.000 }
gfCNCPoint2[20762] = {X 442.2903, Y 47.5438, Z -3.0000, A 0.000, B 0.000, C 0.000 }
gfCNCPoint2[20763] = {X 441.6443, Y 48.1899, Z -3.0000, A 0.000, B 0.000, C 0.000 }
gfCNCPoint2[20764] = {X 440.8707, Y 48.6760, Z -3.0000, A 0.000, B 0.000, C 0.000 }
gfCNCPoint2[20765] = {X 440.0084, Y 48.9777, Z -3.0000, A 0.000, B 0.000, C 0.000 }
gfCNCPoint2[20766] = {X 439.1005, Y 49.0800, Z -3.0000, A 0.000, B 0.000, C 0.000 }
gfCNCPoint2[20767] = {X 432.5144, Y 49.0800, Z -3.0000, A 0.000, B 0.000, C 0.000 }
gfCNCPoint2[20768] = {X 431.6065, Y 48.9777, Z -3.0000, A 0.000, B 0.000, C 0.000 }
gfCNCPoint2[20769] = {X 430.7442, Y 48.6760, Z -3.0000, A 0.000, B 0.000, C 0.000 }
gfCNCPoint2[20770] = {X 429.9706, Y 48.1899, Z -3.0000, A 0.000, B 0.000, C 0.000 }
gfCNCPoint2[20771] = {X 429.3245, Y 47.5438, Z -3.0000, A 0.000, B 0.000, C 0.000 }
gfCNCPoint2[20772] = {X 428.8385, Y 46.7702, Z -3.0000, A 0.000, B 0.000, C 0.000 }
gfCNCPoint2[20773] = {X 428.5367, Y 45.9079, Z -3.0000, A 0.000, B 0.000, C 0.000 }
gfCNCPoint2[20774] = {X 428.4344, Y 45.0000, Z -3.0000, A 0.000, B 0.000, C 0.000 }
gfCNCPoint2[20775] = {X 428.4348, Y 44.1527, Z -3.0000, A 0.000, B 0.000, C 0.000 }
gfCNCPoint2[20776] = {X 428.5303, Y 43.3294, Z -3.0000, A 0.000, B 0.000, C 0.000 }
gfCNCPoint2[20777] = {X 428.7902, Y 42.5424, Z -3.0000, A 0.000, B 0.000, C 0.000 }
gfCNCPoint2[20778] = {X 429.2038, Y 41.8242, Z -3.0000, A 0.000, B 0.000, C 0.000 }
gfCNCPoint2[20779] = {X 429.7540, Y 41.2044, Z -3.0000, A 0.000, B 0.000, C 0.000 }
gfCNCPoint2[20780] = {X 430.4181, Y 40.7085, Z -3.0000, A 0.000, B 0.000, C 0.000 }
gfCNCPoint2[20781] = {X 431.1687, Y 40.3571, Z -3.0000, A 0.000, B 0.000, C 0.000 }
gfCNCPoint2[20782] = {X 435.3052, Y 32.2605, Z -3.0000, A 0.000, B 0.000, C 0.000 }
gfCNCPoint2[20783] = {X 434.1142, Y 31.4918, Z -3.0000, A 0.000, B 0.000, C 0.000 }
gfCNCPoint2[20784] = {X 433.0312, Y 30.5774, Z -3.0000, A 0.000, B 0.000, C 0.000 }
gfCNCPoint2[20785] = {X 432.0737, Y 29.5322, Z -3.0000, A 0.000, B 0.000, C 0.000 }
gfCNCPoint2[20786] = {X 431.2575, Y 28.3734, Z -3.0000, A 0.000, B 0.000, C 0.000 }
gfCNCPoint2[20787] = {X 430.5958, Y 27.1198, Z -3.0000, A 0.000, B 0.000, C 0.000 }
gfCNCPoint2[20788] = {X 430.0997, Y 25.7920, Z -3.0000, A 0.000, B 0.000, C 0.000 }
gfCNCPoint2[20789] = {X 429.6870, Y 24.0071, Z -3.0000, A 0.000, B 0.000, C 0.000 }
gfCNCPoint2[20790] = {X 429.4767, Y 22.1872, Z -3.0000, A 0.000, B 0.000, C 0.000 }
gfCNCPoint2[20791] = {X 429.4716, Y 20.3552, Z -3.0000, A 0.000, B 0.000, C 0.000 }
gfCNCPoint2[20792] = {X 429.6716, Y 18.5341, Z -3.0000, A 0.000, B 0.000, C 0.000 }
gfCNCPoint2[20793] = {X 430.0742, Y 16.7469, Z -3.0000, A 0.000, B 0.000, C 0.000 }
gfCNCPoint2[20794] = {X 430.5851, Y 15.3070, Z -3.0000, A 0.000, B 0.000, C 0.000 }
gfCNCPoint2[20795] = {X 431.2815, Y 13.9470, Z -3.0000, A 0.000, B 0.000, C 0.000 }
gfCNCPoint2[20796] = {X 432.1512, Y 12.6908, Z -3.0000, A 0.000, B 0.000, C 0.000 }
gfCNCPoint2[20797] = {X 433.1791, Y 11.5604, Z -3.0000, A 0.000, B 0.000, C 0.000 }
gfCNCPoint2[20798] = {X 434.3471, Y 10.5755, Z -3.0000, A 0.000, B 0.000, C 0.000 }
gfCNCPoint2[20799] = {X 435.6349, Y 9.7533, Z -3.0000, A 0.000, B 0.000, C 0.000 }
gfCNCPoint2[20800] = {X 437.0200, Y 9.1083, Z -3.0000, A 0.000, B 0.000, C 0.000 }
gfCNCPoint2[20801] = {X 438.4780, Y 8.6516, Z -3.0000, A 0.000, B 0.000, C 0.000 }
gfCNCPoint2[20802] = {X 440.0845, Y 8.3466, Z -3.0000, A 0.000, B 0.000, C 0.000 }
gfCNCPoint2[20803] = {X 441.7099, Y 8.1674, Z -3.0000, A 0.000, B 0.000, C 0.000 }
gfCNCPoint2[20804] = {X 443.3442, Y 8.1153, Z -3.0000, A 0.000, B 0.000, C 0.000 }
gfCNCPoint2[20805] = {X 444.0364, Y 8.1112, Z -3.0000, A 0.000, B 0.000, C 0.000 }
gfCNCPoint2[20806] = {X 459.4466, Y 8.1112, Z -3.0000, A 0.000, B 0.000, C 0.000 }
gfCNCPoint2[20807] = {X 460.3525, Y 8.2133, Z -3.0000, A 0.000, B 0.000, C 0.000 }
gfCNCPoint2[20808] = {X 461.2131, Y 8.5144, Z -3.0000, A 0.000, B 0.000, C 0.000 }
gfCNCPoint2[20809] = {X 461.9850, Y 8.9995, Z -3.0000, A 0.000, B 0.000, C 0.000 }
gfCNCPoint2[20810] = {X 462.6297, Y 9.6441, Z -3.0000, A 0.000, B 0.000, C 0.000 }
gfCNCPoint2[20811] = {X 463.1148, Y 10.4161, Z -3.0000, A 0.000, B 0.000, C 0.000 }
gfCNCPoint2[20812] = {X 463.4159, Y 11.2766, Z -3.0000, A 0.000, B 0.000, C 0.000 }
gfCNCPoint2[20813] = {X 463.5179, Y 12.1826, Z -3.0000, A 0.000, B 0.000, C 0.000 }
gfCNCPoint2[20814] = {X 463.5179, Y 12.9781, Z -3.0000, A 0.000, B 0.000, C 0.000 }
gfCNCPoint2[20815] = {X 463.4241, Y 13.8482, Z -3.0000, A 0.000, B 0.000, C 0.000 }
gfCNCPoint2[20816] = {X 463.1468, Y 14.6782, Z -3.0000, A 0.000, B 0.000, C 0.000 }
gfCNCPoint2[20817] = {X 462.6989, Y 15.4300, Z -3.0000, A 0.000, B 0.000, C 0.000 }
gfCNCPoint2[20818] = {X 462.1010, Y 16.0691, Z -3.0000, A 0.000, B 0.000, C 0.000 }
gfCNCPoint2[20819] = {X 462.0436, Y 16.1176, Z -3.0000, A 0.000, B 0.000, C 0.000 }
gfCNCPoint2[20820] = {X 461.9854, Y 16.1650, Z -3.0000, A 0.000, B 0.000, C 0.000 }
gfCNCPoint2[20821] = {X 461.9900, Y 16.1995, Z -3.0000, A 0.000, B 0.000, C 0.000 }
gfCNCPoint2[20822] = {X 461.9902, Y 28.5935, Z -3.0000, A 0.000, B 0.000, C 0.000 }
gfCNCPoint2[20823] = {X 465.9902, Y 28.5935, Z -3.0000, A 0.000, B 0.000, C 0.000 }
gfCNCPoint2[20824] = {X 465.9902, Y 28.5934, Z -3.0000, A 0.000, B 0.000, C 0.000 }
gfCNCPoint2[20825] = {X 461.9099, Y 28.5935, Z -3.0000, A 0.000, B 0.000, C 0.000 }
gfCNCPoint2[20826] = {X 461.9105, Y 41.0656, Z -3.0000, A 0.000, B 0.000, C 0.000 }
gfCNCPoint2[20827] = {X 462.0493, Y 41.1788, Z -3.0000, A 0.000, B 0.000, C 0.000 }
gfCNCPoint2[20828] = {X 462.6353, Y 41.8053, Z -3.0000, A 0.000, B 0.000, C 0.000 }
gfCNCPoint2[20829] = {X 463.0743, Y 42.5423, Z -3.0000, A 0.000, B 0.000, C 0.000 }
gfCNCPoint2[20830] = {X 463.3460, Y 43.3560, Z -3.0000, A 0.000, B 0.000, C 0.000 }
gfCNCPoint2[20831] = {X 463.4379, Y 44.2089, Z -3.0000, A 0.000, B 0.000, C 0.000 }
gfCNCPoint2[20832] = {X 463.4379, Y 45.0000, Z -3.0000, A 0.000, B 0.000, C 0.000 }
gfCNCPoint2[20833] = {X 463.3377, Y 45.8901, Z -3.0000, A 0.000, B 0.000, C 0.000 }
gfCNCPoint2[20834] = {X 463.0418, Y 46.7355, Z -3.0000, A 0.000, B 0.000, C 0.000 }
gfCNCPoint2[20835] = {X 462.5653, Y 47.4940, Z -3.0000, A 0.000, B 0.000, C 0.000 }
gfCNCPoint2[20836] = {X 461.9319, Y 48.1273, Z -3.0000, A 0.000, B 0.000, C 0.000 }
gfCNCPoint2[20837] = {X 461.1735, Y 48.6039, Z -3.0000, A 0.000, B 0.000, C 0.000 }
gfCNCPoint2[20838] = {X 460.3280, Y 48.8997, Z -3.0000, A 0.000, B 0.000, C 0.000 }
gfCNCPoint2[20839] = {X 459.4379, Y 49.0000, Z -3.0000, A 0.000, B 0.000, C 0.000 }
gfCNCPoint2[20840] = {X 452.9945, Y 49.0000, Z -3.0000, A 0.000, B 0.000, C 0.000 }
gfCNCPoint2[20841] = {X 452.1044, Y 48.8997, Z -3.0000, A 0.000, B 0.000, C 0.000 }
gfCNCPoint2[20842] = {X 451.2589, Y 48.6039, Z -3.0000, A 0.000, B 0.000, C 0.000 }
gfCNCPoint2[20843] = {X 450.5005, Y 48.1273, Z -3.0000, A 0.000, B 0.000, C 0.000 }
gfCNCPoint2[20844] = {X 449.8671, Y 47.4939, Z -3.0000, A 0.000, B 0.000, C 0.000 }
gfCNCPoint2[20845] = {X 449.3906, Y 46.7355, Z -3.0000, A 0.000, B 0.000, C 0.000 }
gfCNCPoint2[20846] = {X 449.0948, Y 45.8900, Z -3.0000, A 0.000, B 0.000, C 0.000 }
gfCNCPoint2[20847] = {X 448.9945, Y 45.0000, Z -3.0000, A 0.000, B 0.000, C 0.000 }
gfCNCPoint2[20848] = {X 448.9949, Y 44.1538, Z -3.0000, A 0.000, B 0.000, C 0.000 }
gfCNCPoint2[20849] = {X 449.1055, Y 43.2730, Z -3.0000, A 0.000, B 0.000, C 0.000 }
gfCNCPoint2[20850] = {X 449.4077, Y 42.4382, Z -3.0000, A 0.000, B 0.000, C 0.000 }
gfCNCPoint2[20851] = {X 449.8865, Y 41.6907, Z -3.0000, A 0.000, B 0.000, C 0.000 }
gfCNCPoint2[20852] = {X 450.5184, Y 41.0672, Z -3.0000, A 0.000, B 0.000, C 0.000 }
gfCNCPoint2[20853] = {X 450.5184, Y 34.1538, Z -3.0000, A 0.000, B 0.000, C 0.000 }
gfCNCPoint2[20854] = {X 447.5228, Y 34.1538, Z -3.0000, A 0.000, B 0.000, C 0.000 }
gfCNCPoint2[20855] = {X 447.2792, Y 34.1526, Z -3.0000, A 0.000, B 0.000, C 0.000 }
gfCNCPoint2[20856] = {X 442.8403, Y 42.7951, Z -3.0000, A 0.000, B 0.000, C 0.000 }
gfCNCPoint2[20857] = {X 442.8966, Y 42.9480, Z -3.0000, A 0.000, B 0.000, C 0.000 }
gfCNCPoint2[20858] = {X 443.0492, Y 43.5703, Z -3.0000, A 0.000, B 0.000, C 0.000 }
gfCNCPoint2[20859] = {X 443.1005, Y 44.2089, Z -3.0000, A 0.000, B 0.000, C 0.000 }
gfCNCPoint2[20860] = {X 443.1005, Y 45.0000, Z -3.0000, A 0.000, B 0.000, C 0.000 }
gfCNCPoint2[20861] = {X 443.0002, Y 45.8901, Z -3.0000, A 0.000, B 0.000, C 0.000 }
gfCNCPoint2[20862] = {X 442.7043, Y 46.7355, Z -3.0000, A 0.000, B 0.000, C 0.000 }
gfCNCPoint2[20863] = {X 442.2278, Y 47.4940, Z -3.0000, A 0.000, B 0.000, C 0.000 }
gfCNCPoint2[20864] = {X 441.5944, Y 48.1273, Z -3.0000, A 0.000, B 0.000, C 0.000 }
gfCNCPoint2[20865] = {X 440.8360, Y 48.6039, Z -3.0000, A 0.000, B 0.000, C 0.000 }
gfCNCPoint2[20866] = {X 439.9906, Y 48.8997, Z -3.0000, A 0.000, B 0.000, C 0.000 }
gfCNCPoint2[20867] = {X 439.1005, Y 49.0000, Z -3.0000, A 0.000, B 0.000, C 0.000 }
gfCNCPoint2[20868] = {X 432.5144, Y 49.0000, Z -3.0000, A 0.000, B 0.000, C 0.000 }
gfCNCPoint2[20869] = {X 431.6243, Y 48.8997, Z -3.0000, A 0.000, B 0.000, C 0.000 }
gfCNCPoint2[20870] = {X 430.7789, Y 48.6039, Z -3.0000, A 0.000, B 0.000, C 0.000 }
gfCNCPoint2[20871] = {X 430.0204, Y 48.1273, Z -3.0000, A 0.000, B 0.000, C 0.000 }
gfCNCPoint2[20872] = {X 429.3871, Y 47.4940, Z -3.0000, A 0.000, B 0.000, C 0.000 }
gfCNCPoint2[20873] = {X 428.9105, Y 46.7355, Z -3.0000, A 0.000, B 0.000, C 0.000 }
gfCNCPoint2[20874] = {X 428.6147, Y 45.8901, Z -3.0000, A 0.000, B 0.000, C 0.000 }
gfCNCPoint2[20875] = {X 428.5144, Y 45.0000, Z -3.0000, A 0.000, B 0.000, C 0.000 }
gfCNCPoint2[20876] = {X 428.5148, Y 44.1538, Z -3.0000, A 0.000, B 0.000, C 0.000 }
gfCNCPoint2[20877] = {X 428.6096, Y 43.3414, Z -3.0000, A 0.000, B 0.000, C 0.000 }
gfCNCPoint2[20878] = {X 428.8676, Y 42.5654, Z -3.0000, A 0.000, B 0.000, C 0.000 }
gfCNCPoint2[20879] = {X 429.2781, Y 41.8580, Z -3.0000, A 0.000, B 0.000, C 0.000 }
gfCNCPoint2[20880] = {X 429.8239, Y 41.2489, Z -3.0000, A 0.000, B 0.000, C 0.000 }
gfCNCPoint2[20881] = {X 430.4821, Y 40.7635, Z -3.0000, A 0.000, B 0.000, C 0.000 }
gfCNCPoint2[20882] = {X 431.2253, Y 40.4222, Z -3.0000, A 0.000, B 0.000, C 0.000 }
gfCNCPoint2[20883] = {X 435.4116, Y 32.2280, Z -3.0000, A 0.000, B 0.000, C 0.000 }
gfCNCPoint2[20884] = {X 434.2136, Y 31.4656, Z -3.0000, A 0.000, B 0.000, C 0.000 }
gfCNCPoint2[20885] = {X 433.1237, Y 30.5552, Z -3.0000, A 0.000, B 0.000, C 0.000 }
gfCNCPoint2[20886] = {X 432.1602, Y 29.5121, Z -3.0000, A 0.000, B 0.000, C 0.000 }
gfCNCPoint2[20887] = {X 431.3391, Y 28.3535, Z -3.0000, A 0.000, B 0.000, C 0.000 }
gfCNCPoint2[20888] = {X 430.6741, Y 27.0988, Z -3.0000, A 0.000, B 0.000, C 0.000 }
gfCNCPoint2[20889] = {X 430.1762, Y 25.7689, Z -3.0000, A 0.000, B 0.000, C 0.000 }
gfCNCPoint2[20890] = {X 429.7657, Y 23.9928, Z -3.0000, A 0.000, B 0.000, C 0.000 }
gfCNCPoint2[20891] = {X 429.5565, Y 22.1819, Z -3.0000, A 0.000, B 0.000, C 0.000 }
gfCNCPoint2[20892] = {X 429.5515, Y 20.3591, Z -3.0000, A 0.000, B 0.000, C 0.000 }
gfCNCPoint2[20893] = {X 429.7505, Y 18.5471, Z -3.0000, A 0.000, B 0.000, C 0.000 }
gfCNCPoint2[20894] = {X 430.1512, Y 16.7687, Z -3.0000, A 0.000, B 0.000, C 0.000 }
gfCNCPoint2[20895] = {X 430.6585, Y 15.3387, Z -3.0000, A 0.000, B 0.000, C 0.000 }
gfCNCPoint2[20896] = {X 431.3500, Y 13.9882, Z -3.0000, A 0.000, B 0.000, C 0.000 }
gfCNCPoint2[20897] = {X 432.2138, Y 12.7407, Z -3.0000, A 0.000, B 0.000, C 0.000 }
gfCNCPoint2[20898] = {X 433.2345, Y 11.6181, Z -3.0000, A 0.000, B 0.000, C 0.000 }
gfCNCPoint2[20899] = {X 434.3945, Y 10.6400, Z -3.0000, A 0.000, B 0.000, C 0.000 }
gfCNCPoint2[20900] = {X 435.6734, Y 9.8235, Z -3.0000, A 0.000, B 0.000, C 0.000 }
gfCNCPoint2[20901] = {X 437.0488, Y 9.1829, Z -3.0000, A 0.000, B 0.000, C 0.000 }
gfCNCPoint2[20902] = {X 438.4968, Y 8.7294, Z -3.0000, A 0.000, B 0.000, C 0.000 }
gfCNCPoint2[20903] = {X 440.0971, Y 8.4256, Z -3.0000, A 0.000, B 0.000, C 0.000 }
gfCNCPoint2[20904] = {X 441.7161, Y 8.2472, Z -3.0000, A 0.000, B 0.000, C 0.000 }
gfCNCPoint2[20905] = {X 443.3442, Y 8.1953, Z -3.0000, A 0.000, B 0.000, C 0.000 }
gfCNCPoint2[20906] = {X 444.0367, Y 8.1912, Z -3.0000, A 0.000, B 0.000, C 0.000 }
gfCNCPoint2[20907] = {X 459.4466, Y 8.1912, Z -3.0000, A 0.000, B 0.000, C 0.000 }
gfCNCPoint2[20908] = {X 460.3347, Y 8.2913, Z -3.0000, A 0.000, B 0.000, C 0.000 }
gfCNCPoint2[20909] = {X 461.1784, Y 8.5865, Z -3.0000, A 0.000, B 0.000, C 0.000 }
gfCNCPoint2[20910] = {X 461.9352, Y 9.0620, Z -3.0000, A 0.000, B 0.000, C 0.000 }
gfCNCPoint2[20911] = {X 462.5672, Y 9.6940, Z -3.0000, A 0.000, B 0.000, C 0.000 }
gfCNCPoint2[20912] = {X 463.0427, Y 10.4508, Z -3.0000, A 0.000, B 0.000, C 0.000 }
gfCNCPoint2[20913] = {X 463.3379, Y 11.2944, Z -3.0000, A 0.000, B 0.000, C 0.000 }
gfCNCPoint2[20914] = {X 463.4379, Y 12.1826, Z -3.0000, A 0.000, B 0.000, C 0.000 }
gfCNCPoint2[20915] = {X 463.4378, Y 13.0163, Z -3.0000, A 0.000, B 0.000, C 0.000 }
gfCNCPoint2[20916] = {X 463.3397, Y 13.8591, Z -3.0000, A 0.000, B 0.000, C 0.000 }
gfCNCPoint2[20917] = {X 463.0661, Y 14.6622, Z -3.0000, A 0.000, B 0.000, C 0.000 }
gfCNCPoint2[20918] = {X 462.6292, Y 15.3896, Z -3.0000, A 0.000, B 0.000, C 0.000 }
gfCNCPoint2[20919] = {X 462.0488, Y 16.0084, Z -3.0000, A 0.000, B 0.000, C 0.000 }
gfCNCPoint2[20920] = {X 461.9723, Y 16.0727, Z -3.0000, A 0.000, B 0.000, C 0.000 }
gfCNCPoint2[20921] = {X 461.8942, Y 16.1351, Z -3.0000, A 0.000, B 0.000, C 0.000 }
gfCNCPoint2[20922] = {X 461.9100, Y 16.1927, Z -3.0000, A 0.000, B 0.000, C 0.000 }
gfCNCPoint2[20923] = {X 461.9093, Y 16.7687, Z -3.0000, A 0.000, B 0.000, C 0.000 }
gfCNCPoint2[20924] = {X 461.9099, Y 28.5935, Z -3.0000, A 0.000, B 0.000, C 0.000 }
gfCNCPoint2[20925] = {X 465.9902, Y 28.5934, Z -3.0000, A 0.000, B 0.000, C 0.000 }
gfCNCPoint2[20926] = {X 465.9902, Y 28.5934, Z 0.0000, A 0.000, B 0.000, C 0.000 }
gfCNCPoint2[20927] = {X 465.9902, Y 28.5934, Z 11.0000, A 0.000, B 0.000, C 0.000 }
gfCNCPoint2[20928] = {X 492.3825, Y 3.7912, Z 11.0000, A 0.000, B 0.000, C 0.000 }
gfCNCPoint2[20929] = {X 492.3825, Y 3.7912, Z 0.0000, A 0.000, B 0.000, C 0.000 }
gfCNCPoint2[20930] = {X 492.3825, Y 3.7912, Z -3.0000, A 0.000, B 0.000, C 0.000 }
gfCNCPoint2[20931] = {X 492.3825, Y 7.8712, Z -3.0000, A 0.000, B 0.000, C 0.000 }
gfCNCPoint2[20932] = {X 502.2066, Y 7.8712, Z -3.0000, A 0.000, B 0.000, C 0.000 }
gfCNCPoint2[20933] = {X 502.7374, Y 7.8754, Z -3.0000, A 0.000, B 0.000, C 0.000 }
gfCNCPoint2[20934] = {X 503.6897, Y 7.9897, Z -3.0000, A 0.000, B 0.000, C 0.000 }
gfCNCPoint2[20935] = {X 504.5931, Y 8.3120, Z -3.0000, A 0.000, B 0.000, C 0.000 }
gfCNCPoint2[20936] = {X 505.4027, Y 8.8264, Z -3.0000, A 0.000, B 0.000, C 0.000 }
gfCNCPoint2[20937] = {X 506.0783, Y 9.5073, Z -3.0000, A 0.000, B 0.000, C 0.000 }
gfCNCPoint2[20938] = {X 506.5863, Y 10.3209, Z -3.0000, A 0.000, B 0.000, C 0.000 }
gfCNCPoint2[20939] = {X 506.9016, Y 11.2268, Z -3.0000, A 0.000, B 0.000, C 0.000 }
gfCNCPoint2[20940] = {X 507.0085, Y 12.1800, Z -3.0000, A 0.000, B 0.000, C 0.000 }
gfCNCPoint2[20941] = {X 507.0085, Y 12.9781, Z -3.0000, A 0.000, B 0.000, C 0.000 }
gfCNCPoint2[20942] = {X 506.9071, Y 13.9083, Z -3.0000, A 0.000, B 0.000, C 0.000 }
gfCNCPoint2[20943] = {X 506.6079, Y 14.7947, Z -3.0000, A 0.000, B 0.000, C 0.000 }
gfCNCPoint2[20944] = {X 506.1248, Y 15.5960, Z -3.0000, A 0.000, B 0.000, C 0.000 }
gfCNCPoint2[20945] = {X 505.4806, Y 16.2745, Z -3.0000, A 0.000, B 0.000, C 0.000 }
gfCNCPoint2[20946] = {X 505.4805, Y 40.9123, Z -3.0000, A 0.000, B 0.000, C 0.000 }
gfCNCPoint2[20947] = {X 506.1191, Y 41.5833, Z -3.0000, A 0.000, B 0.000, C 0.000 }
gfCNCPoint2[20948] = {X 506.6000, Y 42.3751, Z -3.0000, A 0.000, B 0.000, C 0.000 }
gfCNCPoint2[20949] = {X 506.9010, Y 43.2512, Z -3.0000, A 0.000, B 0.000, C 0.000 }
gfCNCPoint2[20950] = {X 507.0083, Y 44.1713, Z -3.0000, A 0.000, B 0.000, C 0.000 }
gfCNCPoint2[20951] = {X 507.0085, Y 45.0000, Z -3.0000, A 0.000, B 0.000, C 0.000 }
gfCNCPoint2[20952] = {X 506.9002, Y 45.9613, Z -3.0000, A 0.000, B 0.000, C 0.000 }
gfCNCPoint2[20953] = {X 506.5807, Y 46.8744, Z -3.0000, A 0.000, B 0.000, C 0.000 }
gfCNCPoint2[20954] = {X 506.0660, Y 47.6935, Z -3.0000, A 0.000, B 0.000, C 0.000 }
gfCNCPoint2[20955] = {X 505.3820, Y 48.3775, Z -3.0000, A 0.000, B 0.000, C 0.000 }
gfCNCPoint2[20956] = {X 504.5629, Y 48.8922, Z -3.0000, A 0.000, B 0.000, C 0.000 }
gfCNCPoint2[20957] = {X 503.6498, Y 49.2117, Z -3.0000, A 0.000, B 0.000, C 0.000 }
gfCNCPoint2[20958] = {X 502.6885, Y 49.3200, Z -3.0000, A 0.000, B 0.000, C 0.000 }
gfCNCPoint2[20959] = {X 496.2450, Y 49.3200, Z -3.0000, A 0.000, B 0.000, C 0.000 }
gfCNCPoint2[20960] = {X 495.2885, Y 49.2128, Z -3.0000, A 0.000, B 0.000, C 0.000 }
gfCNCPoint2[20961] = {X 494.3794, Y 48.8964, Z -3.0000, A 0.000, B 0.000, C 0.000 }
gfCNCPoint2[20962] = {X 493.5630, Y 48.3866, Z -3.0000, A 0.000, B 0.000, C 0.000 }
gfCNCPoint2[20963] = {X 492.8797, Y 47.7087, Z -3.0000, A 0.000, B 0.000, C 0.000 }
gfCNCPoint2[20964] = {X 492.3635, Y 46.8963, Z -3.0000, A 0.000, B 0.000, C 0.000 }
gfCNCPoint2[20965] = {X 492.0399, Y 45.9898, Z -3.0000, A 0.000, B 0.000, C 0.000 }
gfCNCPoint2[20966] = {X 491.9252, Y 45.0341, Z -3.0000, A 0.000, B 0.000, C 0.000 }
gfCNCPoint2[20967] = {X 491.9254, Y 44.1494, Z -3.0000, A 0.000, B 0.000, C 0.000 }
gfCNCPoint2[20968] = {X 492.0359, Y 43.2364, Z -3.0000, A 0.000, B 0.000, C 0.000 }
gfCNCPoint2[20969] = {X 492.3371, Y 42.3675, Z -3.0000, A 0.000, B 0.000, C 0.000 }
gfCNCPoint2[20970] = {X 492.8153, Y 41.5821, Z -3.0000, A 0.000, B 0.000, C 0.000 }
gfCNCPoint2[20971] = {X 493.4490, Y 40.9157, Z -3.0000, A 0.000, B 0.000, C 0.000 }
gfCNCPoint2[20972] = {X 493.4490, Y 34.4738, Z -3.0000, A 0.000, B 0.000, C 0.000 }
gfCNCPoint2[20973] = {X 490.7238, Y 34.4738, Z -3.0000, A 0.000, B 0.000, C 0.000 }
gfCNCPoint2[20974] = {X 486.4398, Y 42.8161, Z -3.0000, A 0.000, B 0.000, C 0.000 }
gfCNCPoint2[20975] = {X 486.4448, Y 42.8293, Z -3.0000, A 0.000, B 0.000, C 0.000 }
gfCNCPoint2[20976] = {X 486.6109, Y 43.4906, Z -3.0000, A 0.000, B 0.000, C 0.000 }
gfCNCPoint2[20977] = {X 486.6708, Y 44.1699, Z -3.0000, A 0.000, B 0.000, C 0.000 }
gfCNCPoint2[20978] = {X 486.6710, Y 45.0000, Z -3.0000, A 0.000, B 0.000, C 0.000 }
gfCNCPoint2[20979] = {X 486.5627, Y 45.9613, Z -3.0000, A 0.000, B 0.000, C 0.000 }
gfCNCPoint2[20980] = {X 486.2432, Y 46.8744, Z -3.0000, A 0.000, B 0.000, C 0.000 }
gfCNCPoint2[20981] = {X 485.7285, Y 47.6935, Z -3.0000, A 0.000, B 0.000, C 0.000 }
gfCNCPoint2[20982] = {X 485.0445, Y 48.3775, Z -3.0000, A 0.000, B 0.000, C 0.000 }
gfCNCPoint2[20983] = {X 484.2254, Y 48.8922, Z -3.0000, A 0.000, B 0.000, C 0.000 }
gfCNCPoint2[20984] = {X 483.3123, Y 49.2117, Z -3.0000, A 0.000, B 0.000, C 0.000 }
gfCNCPoint2[20985] = {X 482.3510, Y 49.3200, Z -3.0000, A 0.000, B 0.000, C 0.000 }
gfCNCPoint2[20986] = {X 475.7650, Y 49.3200, Z -3.0000, A 0.000, B 0.000, C 0.000 }
gfCNCPoint2[20987] = {X 474.8037, Y 49.2117, Z -3.0000, A 0.000, B 0.000, C 0.000 }
gfCNCPoint2[20988] = {X 473.8906, Y 48.8922, Z -3.0000, A 0.000, B 0.000, C 0.000 }
gfCNCPoint2[20989] = {X 473.0715, Y 48.3775, Z -3.0000, A 0.000, B 0.000, C 0.000 }
gfCNCPoint2[20990] = {X 472.3875, Y 47.6935, Z -3.0000, A 0.000, B 0.000, C 0.000 }
gfCNCPoint2[20991] = {X 471.8728, Y 46.8744, Z -3.0000, A 0.000, B 0.000, C 0.000 }
gfCNCPoint2[20992] = {X 471.5533, Y 45.9614, Z -3.0000, A 0.000, B 0.000, C 0.000 }
gfCNCPoint2[20993] = {X 471.4450, Y 45.0001, Z -3.0000, A 0.000, B 0.000, C 0.000 }
gfCNCPoint2[20994] = {X 471.4454, Y 44.1494, Z -3.0000, A 0.000, B 0.000, C 0.000 }
gfCNCPoint2[20995] = {X 471.5430, Y 43.2935, Z -3.0000, A 0.000, B 0.000, C 0.000 }
gfCNCPoint2[20996] = {X 471.8086, Y 42.4740, Z -3.0000, A 0.000, B 0.000, C 0.000 }
gfCNCPoint2[20997] = {X 472.2314, Y 41.7236, Z -3.0000, A 0.000, B 0.000, C 0.000 }
gfCNCPoint2[20998] = {X 472.7947, Y 41.0719, Z -3.0000, A 0.000, B 0.000, C 0.000 }
gfCNCPoint2[20999] = {X 473.4762, Y 40.5449, Z -3.0000, A 0.000, B 0.000, C 0.000 }
gfCNCPoint2[21000] = {X 474.2486, Y 40.1637, Z -3.0000, A 0.000, B 0.000, C 0.000 }
gfCNCPoint2[21001] = {X 478.2331, Y 32.3645, Z -3.0000, A 0.000, B 0.000, C 0.000 }
gfCNCPoint2[21002] = {X 476.9697, Y 31.4967, Z -3.0000, A 0.000, B 0.000, C 0.000 }
gfCNCPoint2[21003] = {X 475.8334, Y 30.4683, Z -3.0000, A 0.000, B 0.000, C 0.000 }
gfCNCPoint2[21004] = {X 474.8443, Y 29.2976, Z -3.0000, A 0.000, B 0.000, C 0.000 }
gfCNCPoint2[21005] = {X 474.0201, Y 28.0054, Z -3.0000, A 0.000, B 0.000, C 0.000 }
gfCNCPoint2[21006] = {X 473.3755, Y 26.6149, Z -3.0000, A 0.000, B 0.000, C 0.000 }
gfCNCPoint2[21007] = {X 472.9221, Y 25.1508, Z -3.0000, A 0.000, B 0.000, C 0.000 }
gfCNCPoint2[21008] = {X 472.6084, Y 23.4678, Z -3.0000, A 0.000, B 0.000, C 0.000 }
gfCNCPoint2[21009] = {X 472.4682, Y 21.7615, Z -3.0000, A 0.000, B 0.000, C 0.000 }
gfCNCPoint2[21010] = {X 472.5029, Y 20.0498, Z -3.0000, A 0.000, B 0.000, C 0.000 }
gfCNCPoint2[21011] = {X 472.7122, Y 18.3505, Z -3.0000, A 0.000, B 0.000, C 0.000 }
gfCNCPoint2[21012] = {X 473.0938, Y 16.6816, Z -3.0000, A 0.000, B 0.000, C 0.000 }
gfCNCPoint2[21013] = {X 473.6364, Y 15.1667, Z -3.0000, A 0.000, B 0.000, C 0.000 }
gfCNCPoint2[21014] = {X 474.3796, Y 13.7396, Z -3.0000, A 0.000, B 0.000, C 0.000 }
gfCNCPoint2[21015] = {X 475.3096, Y 12.4265, Z -3.0000, A 0.000, B 0.000, C 0.000 }
gfCNCPoint2[21016] = {X 476.4092, Y 11.2517, Z -3.0000, A 0.000, B 0.000, C 0.000 }
gfCNCPoint2[21017] = {X 477.6580, Y 10.2371, Z -3.0000, A 0.000, B 0.000, C 0.000 }
gfCNCPoint2[21018] = {X 479.0331, Y 9.4014, Z -3.0000, A 0.000, B 0.000, C 0.000 }
gfCNCPoint2[21019] = {X 480.5088, Y 8.7600, Z -3.0000, A 0.000, B 0.000, C 0.000 }
gfCNCPoint2[21020] = {X 482.0579, Y 8.3249, Z -3.0000, A 0.000, B 0.000, C 0.000 }
gfCNCPoint2[21021] = {X 484.1552, Y 7.9979, Z -3.0000, A 0.000, B 0.000, C 0.000 }
gfCNCPoint2[21022] = {X 486.2747, Y 7.8834, Z -3.0000, A 0.000, B 0.000, C 0.000 }
gfCNCPoint2[21023] = {X 486.9679, Y 7.8712, Z -3.0000, A 0.000, B 0.000, C 0.000 }
gfCNCPoint2[21024] = {X 492.3825, Y 7.8712, Z -3.0000, A 0.000, B 0.000, C 0.000 }
gfCNCPoint2[21025] = {X 492.3825, Y 3.8712, Z -3.0000, A 0.000, B 0.000, C 0.000 }
gfCNCPoint2[21026] = {X 492.3825, Y 7.9512, Z -3.0000, A 0.000, B 0.000, C 0.000 }
gfCNCPoint2[21027] = {X 502.2063, Y 7.9512, Z -3.0000, A 0.000, B 0.000, C 0.000 }
gfCNCPoint2[21028] = {X 502.7368, Y 7.9554, Z -3.0000, A 0.000, B 0.000, C 0.000 }
gfCNCPoint2[21029] = {X 503.6714, Y 8.0676, Z -3.0000, A 0.000, B 0.000, C 0.000 }
gfCNCPoint2[21030] = {X 504.5580, Y 8.3839, Z -3.0000, A 0.000, B 0.000, C 0.000 }
gfCNCPoint2[21031] = {X 505.3526, Y 8.8887, Z -3.0000, A 0.000, B 0.000, C 0.000 }
gfCNCPoint2[21032] = {X 506.0156, Y 9.5570, Z -3.0000, A 0.000, B 0.000, C 0.000 }
gfCNCPoint2[21033] = {X 506.5142, Y 10.3554, Z -3.0000, A 0.000, B 0.000, C 0.000 }
gfCNCPoint2[21034] = {X 506.8236, Y 11.2445, Z -3.0000, A 0.000, B 0.000, C 0.000 }
gfCNCPoint2[21035] = {X 506.9285, Y 12.1800, Z -3.0000, A 0.000, B 0.000, C 0.000 }
gfCNCPoint2[21036] = {X 506.9285, Y 12.9781, Z -3.0000, A 0.000, B 0.000, C 0.000 }
gfCNCPoint2[21037] = {X 506.8270, Y 13.9000, Z -3.0000, A 0.000, B 0.000, C 0.000 }
gfCNCPoint2[21038] = {X 506.5275, Y 14.7778, Z -3.0000, A 0.000, B 0.000, C 0.000 }
gfCNCPoint2[21039] = {X 506.0444, Y 15.5695, Z -3.0000, A 0.000, B 0.000, C 0.000 }
gfCNCPoint2[21040] = {X 505.4006, Y 16.2372, Z -3.0000, A 0.000, B 0.000, C 0.000 }
gfCNCPoint2[21041] = {X 505.4005, Y 40.9503, Z -3.0000, A 0.000, B 0.000, C 0.000 }
gfCNCPoint2[21042] = {X 505.4288, Y 40.9733, Z -3.0000, A 0.000, B 0.000, C 0.000 }
gfCNCPoint2[21043] = {X 506.0556, Y 41.6320, Z -3.0000, A 0.000, B 0.000, C 0.000 }
gfCNCPoint2[21044] = {X 506.5276, Y 42.4091, Z -3.0000, A 0.000, B 0.000, C 0.000 }
gfCNCPoint2[21045] = {X 506.8230, Y 43.2689, Z -3.0000, A 0.000, B 0.000, C 0.000 }
gfCNCPoint2[21046] = {X 506.9283, Y 44.1720, Z -3.0000, A 0.000, B 0.000, C 0.000 }
gfCNCPoint2[21047] = {X 506.9285, Y 45.0000, Z -3.0000, A 0.000, B 0.000, C 0.000 }
gfCNCPoint2[21048] = {X 506.8222, Y 45.9435, Z -3.0000, A 0.000, B 0.000, C 0.000 }
gfCNCPoint2[21049] = {X 506.5086, Y 46.8397, Z -3.0000, A 0.000, B 0.000, C 0.000 }
gfCNCPoint2[21050] = {X 506.0035, Y 47.6436, Z -3.0000, A 0.000, B 0.000, C 0.000 }
gfCNCPoint2[21051] = {X 505.3321, Y 48.3150, Z -3.0000, A 0.000, B 0.000, C 0.000 }
gfCNCPoint2[21052] = {X 504.5282, Y 48.8201, Z -3.0000, A 0.000, B 0.000, C 0.000 }
gfCNCPoint2[21053] = {X 503.6320, Y 49.1337, Z -3.0000, A 0.000, B 0.000, C 0.000 }
gfCNCPoint2[21054] = {X 502.6885, Y 49.2400, Z -3.0000, A 0.000, B 0.000, C 0.000 }
gfCNCPoint2[21055] = {X 496.2450, Y 49.2400, Z -3.0000, A 0.000, B 0.000, C 0.000 }
gfCNCPoint2[21056] = {X 495.3062, Y 49.1348, Z -3.0000, A 0.000, B 0.000, C 0.000 }
gfCNCPoint2[21057] = {X 494.4140, Y 48.8242, Z -3.0000, A 0.000, B 0.000, C 0.000 }
gfCNCPoint2[21058] = {X 493.6127, Y 48.3239, Z -3.0000, A 0.000, B 0.000, C 0.000 }
gfCNCPoint2[21059] = {X 492.9420, Y 47.6585, Z -3.0000, A 0.000, B 0.000, C 0.000 }
gfCNCPoint2[21060] = {X 492.4354, Y 46.8612, Z -3.0000, A 0.000, B 0.000, C 0.000 }
gfCNCPoint2[21061] = {X 492.1178, Y 45.9714, Z -3.0000, A 0.000, B 0.000, C 0.000 }
gfCNCPoint2[21062] = {X 492.0052, Y 45.0335, Z -3.0000, A 0.000, B 0.000, C 0.000 }
gfCNCPoint2[21063] = {X 492.0054, Y 44.1505, Z -3.0000, A 0.000, B 0.000, C 0.000 }
gfCNCPoint2[21064] = {X 492.1159, Y 43.2454, Z -3.0000, A 0.000, B 0.000, C 0.000 }
gfCNCPoint2[21065] = {X 492.4173, Y 42.3850, Z -3.0000, A 0.000, B 0.000, C 0.000 }
gfCNCPoint2[21066] = {X 492.8957, Y 41.6088, Z -3.0000, A 0.000, B 0.000, C 0.000 }
gfCNCPoint2[21067] = {X 493.5290, Y 40.9529, Z -3.0000, A 0.000, B 0.000, C 0.000 }
gfCNCPoint2[21068] = {X 493.5290, Y 34.3938, Z -3.0000, A 0.000, B 0.000, C 0.000 }
gfCNCPoint2[21069] = {X 490.6750, Y 34.3938, Z -3.0000, A 0.000, B 0.000, C 0.000 }
gfCNCPoint2[21070] = {X 486.3524, Y 42.8112, Z -3.0000, A 0.000, B 0.000, C 0.000 }
gfCNCPoint2[21071] = {X 486.3695, Y 42.8562, Z -3.0000, A 0.000, B 0.000, C 0.000 }
gfCNCPoint2[21072] = {X 486.5321, Y 43.5047, Z -3.0000, A 0.000, B 0.000, C 0.000 }
gfCNCPoint2[21073] = {X 486.5908, Y 44.1706, Z -3.0000, A 0.000, B 0.000, C 0.000 }
gfCNCPoint2[21074] = {X 486.5910, Y 45.0000, Z -3.0000, A 0.000, B 0.000, C 0.000 }
gfCNCPoint2[21075] = {X 486.4847, Y 45.9435, Z -3.0000, A 0.000, B 0.000, C 0.000 }
gfCNCPoint2[21076] = {X 486.1711, Y 46.8397, Z -3.0000, A 0.000, B 0.000, C 0.000 }
gfCNCPoint2[21077] = {X 485.6660, Y 47.6436, Z -3.0000, A 0.000, B 0.000, C 0.000 }
gfCNCPoint2[21078] = {X 484.9946, Y 48.3150, Z -3.0000, A 0.000, B 0.000, C 0.000 }
gfCNCPoint2[21079] = {X 484.1907, Y 48.8201, Z -3.0000, A 0.000, B 0.000, C 0.000 }
gfCNCPoint2[21080] = {X 483.2945, Y 49.1337, Z -3.0000, A 0.000, B 0.000, C 0.000 }
gfCNCPoint2[21081] = {X 482.3510, Y 49.2400, Z -3.0000, A 0.000, B 0.000, C 0.000 }
gfCNCPoint2[21082] = {X 475.7650, Y 49.2400, Z -3.0000, A 0.000, B 0.000, C 0.000 }
gfCNCPoint2[21083] = {X 474.8215, Y 49.1337, Z -3.0000, A 0.000, B 0.000, C 0.000 }
gfCNCPoint2[21084] = {X 473.9253, Y 48.8201, Z -3.0000, A 0.000, B 0.000, C 0.000 }
gfCNCPoint2[21085] = {X 473.1214, Y 48.3150, Z -3.0000, A 0.000, B 0.000, C 0.000 }
gfCNCPoint2[21086] = {X 472.4500, Y 47.6436, Z -3.0000, A 0.000, B 0.000, C 0.000 }
gfCNCPoint2[21087] = {X 471.9449, Y 46.8397, Z -3.0000, A 0.000, B 0.000, C 0.000 }
gfCNCPoint2[21088] = {X 471.6313, Y 45.9436, Z -3.0000, A 0.000, B 0.000, C 0.000 }
gfCNCPoint2[21089] = {X 471.5250, Y 45.0001, Z -3.0000, A 0.000, B 0.000, C 0.000 }
gfCNCPoint2[21090] = {X 471.5254, Y 44.1505, Z -3.0000, A 0.000, B 0.000, C 0.000 }
gfCNCPoint2[21091] = {X 471.6223, Y 43.3054, Z -3.0000, A 0.000, B 0.000, C 0.000 }
gfCNCPoint2[21092] = {X 471.8860, Y 42.4967, Z -3.0000, A 0.000, B 0.000, C 0.000 }
gfCNCPoint2[21093] = {X 472.3057, Y 41.7570, Z -3.0000, A 0.000, B 0.000, C 0.000 }
gfCNCPoint2[21094] = {X 472.8647, Y 41.1158, Z -3.0000, A 0.000, B 0.000, C 0.000 }
gfCNCPoint2[21095] = {X 473.5404, Y 40.5992, Z -3.0000, A 0.000, B 0.000, C 0.000 }
gfCNCPoint2[21096] = {X 474.3057, Y 40.2278, Z -3.0000, A 0.000, B 0.000, C 0.000 }
gfCNCPoint2[21097] = {X 478.3386, Y 32.3338, Z -3.0000, A 0.000, B 0.000, C 0.000 }
gfCNCPoint2[21098] = {X 477.0686, Y 31.4726, Z -3.0000, A 0.000, B 0.000, C 0.000 }
gfCNCPoint2[21099] = {X 475.9258, Y 30.4486, Z -3.0000, A 0.000, B 0.000, C 0.000 }
gfCNCPoint2[21100] = {X 474.9310, Y 29.2803, Z -3.0000, A 0.000, B 0.000, C 0.000 }
gfCNCPoint2[21101] = {X 474.1023, Y 27.9889, Z -3.0000, A 0.000, B 0.000, C 0.000 }
gfCNCPoint2[21102] = {X 473.4547, Y 26.5978, Z -3.0000, A 0.000, B 0.000, C 0.000 }
gfCNCPoint2[21103] = {X 472.9999, Y 25.1323, Z -3.0000, A 0.000, B 0.000, C 0.000 }
gfCNCPoint2[21104] = {X 472.6877, Y 23.4572, Z -3.0000, A 0.000, B 0.000, C 0.000 }
gfCNCPoint2[21105] = {X 472.5481, Y 21.7591, Z -3.0000, A 0.000, B 0.000, C 0.000 }
gfCNCPoint2[21106] = {X 472.5827, Y 20.0555, Z -3.0000, A 0.000, B 0.000, C 0.000 }
gfCNCPoint2[21107] = {X 472.7909, Y 18.3644, Z -3.0000, A 0.000, B 0.000, C 0.000 }
gfCNCPoint2[21108] = {X 473.1708, Y 16.7034, Z -3.0000, A 0.000, B 0.000, C 0.000 }
gfCNCPoint2[21109] = {X 473.7097, Y 15.1988, Z -3.0000, A 0.000, B 0.000, C 0.000 }
gfCNCPoint2[21110] = {X 474.4479, Y 13.7813, Z -3.0000, A 0.000, B 0.000, C 0.000 }
gfCNCPoint2[21111] = {X 475.3716, Y 12.4770, Z -3.0000, A 0.000, B 0.000, C 0.000 }
gfCNCPoint2[21112] = {X 476.4637, Y 11.3103, Z -3.0000, A 0.000, B 0.000, C 0.000 }
gfCNCPoint2[21113] = {X 477.7041, Y 10.3025, Z -3.0000, A 0.000, B 0.000, C 0.000 }
gfCNCPoint2[21114] = {X 479.0699, Y 9.4724, Z -3.0000, A 0.000, B 0.000, C 0.000 }
gfCNCPoint2[21115] = {X 480.5356, Y 8.8354, Z -3.0000, A 0.000, B 0.000, C 0.000 }
gfCNCPoint2[21116] = {X 482.0742, Y 8.4032, Z -3.0000, A 0.000, B 0.000, C 0.000 }
gfCNCPoint2[21117] = {X 484.1638, Y 8.0774, Z -3.0000, A 0.000, B 0.000, C 0.000 }
gfCNCPoint2[21118] = {X 486.2756, Y 7.9634, Z -3.0000, A 0.000, B 0.000, C 0.000 }
gfCNCPoint2[21119] = {X 486.9686, Y 7.9512, Z -3.0000, A 0.000, B 0.000, C 0.000 }
gfCNCPoint2[21120] = {X 492.3825, Y 7.9512, Z -3.0000, A 0.000, B 0.000, C 0.000 }
gfCNCPoint2[21121] = {X 492.3825, Y 3.9512, Z -3.0000, A 0.000, B 0.000, C 0.000 }
gfCNCPoint2[21122] = {X 492.3825, Y 8.0312, Z -3.0000, A 0.000, B 0.000, C 0.000 }
gfCNCPoint2[21123] = {X 502.2059, Y 8.0312, Z -3.0000, A 0.000, B 0.000, C 0.000 }
gfCNCPoint2[21124] = {X 502.7361, Y 8.0354, Z -3.0000, A 0.000, B 0.000, C 0.000 }
gfCNCPoint2[21125] = {X 503.6531, Y 8.1454, Z -3.0000, A 0.000, B 0.000, C 0.000 }
gfCNCPoint2[21126] = {X 504.5229, Y 8.4558, Z -3.0000, A 0.000, B 0.000, C 0.000 }
gfCNCPoint2[21127] = {X 505.3024, Y 8.9511, Z -3.0000, A 0.000, B 0.000, C 0.000 }
gfCNCPoint2[21128] = {X 505.9529, Y 9.6066, Z -3.0000, A 0.000, B 0.000, C 0.000 }
gfCNCPoint2[21129] = {X 506.4420, Y 10.3900, Z -3.0000, A 0.000, B 0.000, C 0.000 }
gfCNCPoint2[21130] = {X 506.7456, Y 11.2622, Z -3.0000, A 0.000, B 0.000, C 0.000 }
gfCNCPoint2[21131] = {X 506.8485, Y 12.1800, Z -3.0000, A 0.000, B 0.000, C 0.000 }
gfCNCPoint2[21132] = {X 506.8485, Y 12.9781, Z -3.0000, A 0.000, B 0.000, C 0.000 }
gfCNCPoint2[21133] = {X 506.7469, Y 13.8918, Z -3.0000, A 0.000, B 0.000, C 0.000 }
gfCNCPoint2[21134] = {X 506.4471, Y 14.7608, Z -3.0000, A 0.000, B 0.000, C 0.000 }
gfCNCPoint2[21135] = {X 505.9638, Y 15.5427, Z -3.0000, A 0.000, B 0.000, C 0.000 }
gfCNCPoint2[21136] = {X 505.3206, Y 16.1995, Z -3.0000, A 0.000, B 0.000, C 0.000 }
gfCNCPoint2[21137] = {X 505.3205, Y 40.9887, Z -3.0000, A 0.000, B 0.000, C 0.000 }
gfCNCPoint2[21138] = {X 505.3676, Y 41.0263, Z -3.0000, A 0.000, B 0.000, C 0.000 }
gfCNCPoint2[21139] = {X 505.9864, Y 41.6732, Z -3.0000, A 0.000, B 0.000, C 0.000 }
gfCNCPoint2[21140] = {X 506.4525, Y 42.4374, Z -3.0000, A 0.000, B 0.000, C 0.000 }
gfCNCPoint2[21141] = {X 506.7443, Y 43.2836, Z -3.0000, A 0.000, B 0.000, C 0.000 }
gfCNCPoint2[21142] = {X 506.8483, Y 44.1727, Z -3.0000, A 0.000, B 0.000, C 0.000 }
gfCNCPoint2[21143] = {X 506.8485, Y 45.0000, Z -3.0000, A 0.000, B 0.000, C 0.000 }
gfCNCPoint2[21144] = {X 506.7442, Y 45.9257, Z -3.0000, A 0.000, B 0.000, C 0.000 }
gfCNCPoint2[21145] = {X 506.4365, Y 46.8050, Z -3.0000, A 0.000, B 0.000, C 0.000 }
gfCNCPoint2[21146] = {X 505.9409, Y 47.5937, Z -3.0000, A 0.000, B 0.000, C 0.000 }
gfCNCPoint2[21147] = {X 505.2822, Y 48.2524, Z -3.0000, A 0.000, B 0.000, C 0.000 }
gfCNCPoint2[21148] = {X 504.4934, Y 48.7480, Z -3.0000, A 0.000, B 0.000, C 0.000 }
gfCNCPoint2[21149] = {X 503.6142, Y 49.0557, Z -3.0000, A 0.000, B 0.000, C 0.000 }
gfCNCPoint2[21150] = {X 502.6885, Y 49.1600, Z -3.0000, A 0.000, B 0.000, C 0.000 }
gfCNCPoint2[21151] = {X 496.2450, Y 49.1600, Z -3.0000, A 0.000, B 0.000, C 0.000 }
gfCNCPoint2[21152] = {X 495.3239, Y 49.0567, Z -3.0000, A 0.000, B 0.000, C 0.000 }
gfCNCPoint2[21153] = {X 494.4485, Y 48.7521, Z -3.0000, A 0.000, B 0.000, C 0.000 }
gfCNCPoint2[21154] = {X 493.6623, Y 48.2612, Z -3.0000, A 0.000, B 0.000, C 0.000 }
gfCNCPoint2[21155] = {X 493.0043, Y 47.6084, Z -3.0000, A 0.000, B 0.000, C 0.000 }
gfCNCPoint2[21156] = {X 492.5072, Y 46.8261, Z -3.0000, A 0.000, B 0.000, C 0.000 }
gfCNCPoint2[21157] = {X 492.1957, Y 45.9531, Z -3.0000, A 0.000, B 0.000, C 0.000 }
gfCNCPoint2[21158] = {X 492.0852, Y 45.0328, Z -3.0000, A 0.000, B 0.000, C 0.000 }
gfCNCPoint2[21159] = {X 492.0854, Y 44.1516, Z -3.0000, A 0.000, B 0.000, C 0.000 }
gfCNCPoint2[21160] = {X 492.1960, Y 43.2545, Z -3.0000, A 0.000, B 0.000, C 0.000 }
gfCNCPoint2[21161] = {X 492.4976, Y 42.4026, Z -3.0000, A 0.000, B 0.000, C 0.000 }
gfCNCPoint2[21162] = {X 492.9762, Y 41.6358, Z -3.0000, A 0.000, B 0.000, C 0.000 }
gfCNCPoint2[21163] = {X 493.6090, Y 40.9906, Z -3.0000, A 0.000, B 0.000, C 0.000 }
gfCNCPoint2[21164] = {X 493.6090, Y 34.3138, Z -3.0000, A 0.000, B 0.000, C 0.000 }
gfCNCPoint2[21165] = {X 490.6261, Y 34.3138, Z -3.0000, A 0.000, B 0.000, C 0.000 }
gfCNCPoint2[21166] = {X 486.2650, Y 42.8063, Z -3.0000, A 0.000, B 0.000, C 0.000 }
gfCNCPoint2[21167] = {X 486.2942, Y 42.8832, Z -3.0000, A 0.000, B 0.000, C 0.000 }
gfCNCPoint2[21168] = {X 486.4534, Y 43.5187, Z -3.0000, A 0.000, B 0.000, C 0.000 }
gfCNCPoint2[21169] = {X 486.5108, Y 44.1713, Z -3.0000, A 0.000, B 0.000, C 0.000 }
gfCNCPoint2[21170] = {X 486.5110, Y 45.0000, Z -3.0000, A 0.000, B 0.000, C 0.000 }
gfCNCPoint2[21171] = {X 486.4067, Y 45.9257, Z -3.0000, A 0.000, B 0.000, C 0.000 }
gfCNCPoint2[21172] = {X 486.0990, Y 46.8050, Z -3.0000, A 0.000, B 0.000, C 0.000 }
gfCNCPoint2[21173] = {X 485.6034, Y 47.5937, Z -3.0000, A 0.000, B 0.000, C 0.000 }
gfCNCPoint2[21174] = {X 484.9447, Y 48.2524, Z -3.0000, A 0.000, B 0.000, C 0.000 }
gfCNCPoint2[21175] = {X 484.1560, Y 48.7480, Z -3.0000, A 0.000, B 0.000, C 0.000 }
gfCNCPoint2[21176] = {X 483.2767, Y 49.0557, Z -3.0000, A 0.000, B 0.000, C 0.000 }
gfCNCPoint2[21177] = {X 482.3510, Y 49.1600, Z -3.0000, A 0.000, B 0.000, C 0.000 }
gfCNCPoint2[21178] = {X 475.7650, Y 49.1600, Z -3.0000, A 0.000, B 0.000, C 0.000 }
gfCNCPoint2[21179] = {X 474.8393, Y 49.0557, Z -3.0000, A 0.000, B 0.000, C 0.000 }
gfCNCPoint2[21180] = {X 473.9600, Y 48.7480, Z -3.0000, A 0.000, B 0.000, C 0.000 }
gfCNCPoint2[21181] = {X 473.1713, Y 48.2524, Z -3.0000, A 0.000, B 0.000, C 0.000 }
gfCNCPoint2[21182] = {X 472.5126, Y 47.5937, Z -3.0000, A 0.000, B 0.000, C 0.000 }
gfCNCPoint2[21183] = {X 472.0169, Y 46.8050, Z -3.0000, A 0.000, B 0.000, C 0.000 }
gfCNCPoint2[21184] = {X 471.7093, Y 45.9257, Z -3.0000, A 0.000, B 0.000, C 0.000 }
gfCNCPoint2[21185] = {X 471.6050, Y 45.0000, Z -3.0000, A 0.000, B 0.000, C 0.000 }
gfCNCPoint2[21186] = {X 471.6054, Y 44.1516, Z -3.0000, A 0.000, B 0.000, C 0.000 }
gfCNCPoint2[21187] = {X 471.7016, Y 43.3174, Z -3.0000, A 0.000, B 0.000, C 0.000 }
gfCNCPoint2[21188] = {X 471.9634, Y 42.5195, Z -3.0000, A 0.000, B 0.000, C 0.000 }
gfCNCPoint2[21189] = {X 472.3801, Y 41.7905, Z -3.0000, A 0.000, B 0.000, C 0.000 }
gfCNCPoint2[21190] = {X 472.9347, Y 41.1600, Z -3.0000, A 0.000, B 0.000, C 0.000 }
gfCNCPoint2[21191] = {X 473.6046, Y 40.6537, Z -3.0000, A 0.000, B 0.000, C 0.000 }
gfCNCPoint2[21192] = {X 474.3626, Y 40.2923, Z -3.0000, A 0.000, B 0.000, C 0.000 }
gfCNCPoint2[21193] = {X 478.4444, Y 32.3026, Z -3.0000, A 0.000, B 0.000, C 0.000 }
gfCNCPoint2[21194] = {X 477.1676, Y 31.4483, Z -3.0000, A 0.000, B 0.000, C 0.000 }
gfCNCPoint2[21195] = {X 476.0183, Y 30.4288, Z -3.0000, A 0.000, B 0.000, C 0.000 }
gfCNCPoint2[21196] = {X 475.0178, Y 29.2630, Z -3.0000, A 0.000, B 0.000, C 0.000 }
gfCNCPoint2[21197] = {X 474.1845, Y 27.9724, Z -3.0000, A 0.000, B 0.000, C 0.000 }
gfCNCPoint2[21198] = {X 473.5338, Y 26.5808, Z -3.0000, A 0.000, B 0.000, C 0.000 }
gfCNCPoint2[21199] = {X 473.0777, Y 25.1138, Z -3.0000, A 0.000, B 0.000, C 0.000 }
gfCNCPoint2[21200] = {X 472.7670, Y 23.4467, Z -3.0000, A 0.000, B 0.000, C 0.000 }
gfCNCPoint2[21201] = {X 472.6281, Y 21.7567, Z -3.0000, A 0.000, B 0.000, C 0.000 }
gfCNCPoint2[21202] = {X 472.6625, Y 20.0613, Z -3.0000, A 0.000, B 0.000, C 0.000 }
gfCNCPoint2[21203] = {X 472.8697, Y 18.3782, Z -3.0000, A 0.000, B 0.000, C 0.000 }
gfCNCPoint2[21204] = {X 473.2478, Y 16.7252, Z -3.0000, A 0.000, B 0.000, C 0.000 }
gfCNCPoint2[21205] = {X 473.7830, Y 15.2308, Z -3.0000, A 0.000, B 0.000, C 0.000 }
gfCNCPoint2[21206] = {X 474.5161, Y 13.8230, Z -3.0000, A 0.000, B 0.000, C 0.000 }
gfCNCPoint2[21207] = {X 475.4335, Y 12.5276, Z -3.0000, A 0.000, B 0.000, C 0.000 }
gfCNCPoint2[21208] = {X 476.5183, Y 11.3688, Z -3.0000, A 0.000, B 0.000, C 0.000 }
gfCNCPoint2[21209] = {X 477.7503, Y 10.3679, Z -3.0000, A 0.000, B 0.000, C 0.000 }
gfCNCPoint2[21210] = {X 479.1067, Y 9.5435, Z -3.0000, A 0.000, B 0.000, C 0.000 }
gfCNCPoint2[21211] = {X 480.5624, Y 8.9108, Z -3.0000, A 0.000, B 0.000, C 0.000 }
gfCNCPoint2[21212] = {X 482.0906, Y 8.4815, Z -3.0000, A 0.000, B 0.000, C 0.000 }
gfCNCPoint2[21213] = {X 484.1725, Y 8.1570, Z -3.0000, A 0.000, B 0.000, C 0.000 }
gfCNCPoint2[21214] = {X 486.2765, Y 8.0434, Z -3.0000, A 0.000, B 0.000, C 0.000 }
gfCNCPoint2[21215] = {X 486.9693, Y 8.0312, Z -3.0000, A 0.000, B 0.000, C 0.000 }
gfCNCPoint2[21216] = {X 492.3825, Y 8.0312, Z -3.0000, A 0.000, B 0.000, C 0.000 }
gfCNCPoint2[21217] = {X 492.3825, Y 4.0312, Z -3.0000, A 0.000, B 0.000, C 0.000 }
gfCNCPoint2[21218] = {X 492.3825, Y 8.1112, Z -3.0000, A 0.000, B 0.000, C 0.000 }
gfCNCPoint2[21219] = {X 502.2056, Y 8.1112, Z -3.0000, A 0.000, B 0.000, C 0.000 }
gfCNCPoint2[21220] = {X 502.7355, Y 8.1154, Z -3.0000, A 0.000, B 0.000, C 0.000 }
gfCNCPoint2[21221] = {X 503.6348, Y 8.2233, Z -3.0000, A 0.000, B 0.000, C 0.000 }
gfCNCPoint2[21222] = {X 504.4878, Y 8.5277, Z -3.0000, A 0.000, B 0.000, C 0.000 }
gfCNCPoint2[21223] = {X 505.2522, Y 9.0134, Z -3.0000, A 0.000, B 0.000, C 0.000 }
gfCNCPoint2[21224] = {X 505.8902, Y 9.6563, Z -3.0000, A 0.000, B 0.000, C 0.000 }
gfCNCPoint2[21225] = {X 506.3699, Y 10.4245, Z -3.0000, A 0.000, B 0.000, C 0.000 }
gfCNCPoint2[21226] = {X 506.6676, Y 11.2799, Z -3.0000, A 0.000, B 0.000, C 0.000 }
gfCNCPoint2[21227] = {X 506.7685, Y 12.1800, Z -3.0000, A 0.000, B 0.000, C 0.000 }
gfCNCPoint2[21228] = {X 506.7685, Y 12.9781, Z -3.0000, A 0.000, B 0.000, C 0.000 }
gfCNCPoint2[21229] = {X 506.6668, Y 13.8834, Z -3.0000, A 0.000, B 0.000, C 0.000 }
gfCNCPoint2[21230] = {X 506.3667, Y 14.7436, Z -3.0000, A 0.000, B 0.000, C 0.000 }
gfCNCPoint2[21231] = {X 505.8833, Y 15.5157, Z -3.0000, A 0.000, B 0.000, C 0.000 }
gfCNCPoint2[21232] = {X 505.2406, Y 16.1613, Z -3.0000, A 0.000, B 0.000, C 0.000 }
gfCNCPoint2[21233] = {X 505.2405, Y 41.0272, Z -3.0000, A 0.000, B 0.000, C 0.000 }
gfCNCPoint2[21234] = {X 505.3177, Y 41.0889, Z -3.0000, A 0.000, B 0.000, C 0.000 }
gfCNCPoint2[21235] = {X 505.9239, Y 41.7232, Z -3.0000, A 0.000, B 0.000, C 0.000 }
gfCNCPoint2[21236] = {X 506.3805, Y 42.4724, Z -3.0000, A 0.000, B 0.000, C 0.000 }
gfCNCPoint2[21237] = {X 506.6664, Y 43.3019, Z -3.0000, A 0.000, B 0.000, C 0.000 }
gfCNCPoint2[21238] = {X 506.7683, Y 44.1734, Z -3.0000, A 0.000, B 0.000, C 0.000 }
gfCNCPoint2[21239] = {X 506.7685, Y 45.0000, Z -3.0000, A 0.000, B 0.000, C 0.000 }
gfCNCPoint2[21240] = {X 506.6662, Y 45.9079, Z -3.0000, A 0.000, B 0.000, C 0.000 }
gfCNCPoint2[21241] = {X 506.3644, Y 46.7702, Z -3.0000, A 0.000, B 0.000, C 0.000 }
gfCNCPoint2[21242] = {X 505.8784, Y 47.5438, Z -3.0000, A 0.000, B 0.000, C 0.000 }
gfCNCPoint2[21243] = {X 505.2323, Y 48.1899, Z -3.0000, A 0.000, B 0.000, C 0.000 }
gfCNCPoint2[21244] = {X 504.4587, Y 48.6760, Z -3.0000, A 0.000, B 0.000, C 0.000 }
gfCNCPoint2[21245] = {X 503.5964, Y 48.9777, Z -3.0000, A 0.000, B 0.000, C 0.000 }
gfCNCPoint2[21246] = {X 502.6885, Y 49.0800, Z -3.0000, A 0.000, B 0.000, C 0.000 }
gfCNCPoint2[21247] = {X 496.2450, Y 49.0800, Z -3.0000, A 0.000, B 0.000, C 0.000 }
gfCNCPoint2[21248] = {X 495.3416, Y 48.9787, Z -3.0000, A 0.000, B 0.000, C 0.000 }
gfCNCPoint2[21249] = {X 494.4831, Y 48.6799, Z -3.0000, A 0.000, B 0.000, C 0.000 }
gfCNCPoint2[21250] = {X 493.7120, Y 48.1985, Z -3.0000, A 0.000, B 0.000, C 0.000 }
gfCNCPoint2[21251] = {X 493.0667, Y 47.5582, Z -3.0000, A 0.000, B 0.000, C 0.000 }
gfCNCPoint2[21252] = {X 492.5791, Y 46.7909, Z -3.0000, A 0.000, B 0.000, C 0.000 }
gfCNCPoint2[21253] = {X 492.2736, Y 45.9348, Z -3.0000, A 0.000, B 0.000, C 0.000 }
gfCNCPoint2[21254] = {X 492.1652, Y 45.0322, Z -3.0000, A 0.000, B 0.000, C 0.000 }
gfCNCPoint2[21255] = {X 492.1654, Y 44.1527, Z -3.0000, A 0.000, B 0.000, C 0.000 }
gfCNCPoint2[21256] = {X 492.2760, Y 43.2637, Z -3.0000, A 0.000, B 0.000, C 0.000 }
gfCNCPoint2[21257] = {X 492.5779, Y 42.4203, Z -3.0000, A 0.000, B 0.000, C 0.000 }
gfCNCPoint2[21258] = {X 493.0566, Y 41.6631, Z -3.0000, A 0.000, B 0.000, C 0.000 }
gfCNCPoint2[21259] = {X 493.6890, Y 41.0287, Z -3.0000, A 0.000, B 0.000, C 0.000 }
gfCNCPoint2[21260] = {X 493.6890, Y 34.2338, Z -3.0000, A 0.000, B 0.000, C 0.000 }
gfCNCPoint2[21261] = {X 490.5773, Y 34.2338, Z -3.0000, A 0.000, B 0.000, C 0.000 }
gfCNCPoint2[21262] = {X 486.1776, Y 42.8014, Z -3.0000, A 0.000, B 0.000, C 0.000 }
gfCNCPoint2[21263] = {X 486.2188, Y 42.9101, Z -3.0000, A 0.000, B 0.000, C 0.000 }
gfCNCPoint2[21264] = {X 486.3746, Y 43.5327, Z -3.0000, A 0.000, B 0.000, C 0.000 }
gfCNCPoint2[21265] = {X 486.4309, Y 44.1720, Z -3.0000, A 0.000, B 0.000, C 0.000 }
gfCNCPoint2[21266] = {X 486.4310, Y 45.0000, Z -3.0000, A 0.000, B 0.000, C 0.000 }
gfCNCPoint2[21267] = {X 486.3287, Y 45.9079, Z -3.0000, A 0.000, B 0.000, C 0.000 }
gfCNCPoint2[21268] = {X 486.0270, Y 46.7702, Z -3.0000, A 0.000, B 0.000, C 0.000 }
gfCNCPoint2[21269] = {X 485.5409, Y 47.5438, Z -3.0000, A 0.000, B 0.000, C 0.000 }
gfCNCPoint2[21270] = {X 484.8949, Y 48.1899, Z -3.0000, A 0.000, B 0.000, C 0.000 }
gfCNCPoint2[21271] = {X 484.1213, Y 48.6760, Z -3.0000, A 0.000, B 0.000, C 0.000 }
gfCNCPoint2[21272] = {X 483.2589, Y 48.9777, Z -3.0000, A 0.000, B 0.000, C 0.000 }
gfCNCPoint2[21273] = {X 482.3510, Y 49.0800, Z -3.0000, A 0.000, B 0.000, C 0.000 }
gfCNCPoint2[21274] = {X 475.7650, Y 49.0800, Z -3.0000, A 0.000, B 0.000, C 0.000 }
gfCNCPoint2[21275] = {X 474.8571, Y 48.9777, Z -3.0000, A 0.000, B 0.000, C 0.000 }
gfCNCPoint2[21276] = {X 473.9947, Y 48.6760, Z -3.0000, A 0.000, B 0.000, C 0.000 }
gfCNCPoint2[21277] = {X 473.2211, Y 48.1899, Z -3.0000, A 0.000, B 0.000, C 0.000 }
gfCNCPoint2[21278] = {X 472.5751, Y 47.5438, Z -3.0000, A 0.000, B 0.000, C 0.000 }
gfCNCPoint2[21279] = {X 472.0890, Y 46.7702, Z -3.0000, A 0.000, B 0.000, C 0.000 }
gfCNCPoint2[21280] = {X 471.7873, Y 45.9079, Z -3.0000, A 0.000, B 0.000, C 0.000 }
gfCNCPoint2[21281] = {X 471.6850, Y 45.0000, Z -3.0000, A 0.000, B 0.000, C 0.000 }
gfCNCPoint2[21282] = {X 471.6853, Y 44.1527, Z -3.0000, A 0.000, B 0.000, C 0.000 }
gfCNCPoint2[21283] = {X 471.7809, Y 43.3294, Z -3.0000, A 0.000, B 0.000, C 0.000 }
gfCNCPoint2[21284] = {X 472.0408, Y 42.5424, Z -3.0000, A 0.000, B 0.000, C 0.000 }
gfCNCPoint2[21285] = {X 472.4544, Y 41.8242, Z -3.0000, A 0.000, B 0.000, C 0.000 }
gfCNCPoint2[21286] = {X 473.0046, Y 41.2044, Z -3.0000, A 0.000, B 0.000, C 0.000 }
gfCNCPoint2[21287] = {X 473.6687, Y 40.7085, Z -3.0000, A 0.000, B 0.000, C 0.000 }
gfCNCPoint2[21288] = {X 474.4193, Y 40.3571, Z -3.0000, A 0.000, B 0.000, C 0.000 }
gfCNCPoint2[21289] = {X 478.5504, Y 32.2709, Z -3.0000, A 0.000, B 0.000, C 0.000 }
gfCNCPoint2[21290] = {X 477.2668, Y 31.4236, Z -3.0000, A 0.000, B 0.000, C 0.000 }
gfCNCPoint2[21291] = {X 476.1110, Y 30.4088, Z -3.0000, A 0.000, B 0.000, C 0.000 }
gfCNCPoint2[21292] = {X 475.1047, Y 29.2456, Z -3.0000, A 0.000, B 0.000, C 0.000 }
gfCNCPoint2[21293] = {X 474.2668, Y 27.9558, Z -3.0000, A 0.000, B 0.000, C 0.000 }
gfCNCPoint2[21294] = {X 473.6130, Y 26.5636, Z -3.0000, A 0.000, B 0.000, C 0.000 }
gfCNCPoint2[21295] = {X 473.1555, Y 25.0952, Z -3.0000, A 0.000, B 0.000, C 0.000 }
gfCNCPoint2[21296] = {X 472.8463, Y 23.4362, Z -3.0000, A 0.000, B 0.000, C 0.000 }
gfCNCPoint2[21297] = {X 472.7081, Y 21.7543, Z -3.0000, A 0.000, B 0.000, C 0.000 }
gfCNCPoint2[21298] = {X 472.7423, Y 20.0670, Z -3.0000, A 0.000, B 0.000, C 0.000 }
gfCNCPoint2[21299] = {X 472.9485, Y 18.3921, Z -3.0000, A 0.000, B 0.000, C 0.000 }
gfCNCPoint2[21300] = {X 473.3247, Y 16.7469, Z -3.0000, A 0.000, B 0.000, C 0.000 }
gfCNCPoint2[21301] = {X 473.8563, Y 15.2629, Z -3.0000, A 0.000, B 0.000, C 0.000 }
gfCNCPoint2[21302] = {X 474.5844, Y 13.8646, Z -3.0000, A 0.000, B 0.000, C 0.000 }
gfCNCPoint2[21303] = {X 475.4955, Y 12.5782, Z -3.0000, A 0.000, B 0.000, C 0.000 }
gfCNCPoint2[21304] = {X 476.5728, Y 11.4273, Z -3.0000, A 0.000, B 0.000, C 0.000 }
gfCNCPoint2[21305] = {X 477.7964, Y 10.4333, Z -3.0000, A 0.000, B 0.000, C 0.000 }
gfCNCPoint2[21306] = {X 479.1435, Y 9.6145, Z -3.0000, A 0.000, B 0.000, C 0.000 }
gfCNCPoint2[21307] = {X 480.5893, Y 8.9861, Z -3.0000, A 0.000, B 0.000, C 0.000 }
gfCNCPoint2[21308] = {X 482.1069, Y 8.5598, Z -3.0000, A 0.000, B 0.000, C 0.000 }
gfCNCPoint2[21309] = {X 484.1811, Y 8.2365, Z -3.0000, A 0.000, B 0.000, C 0.000 }
gfCNCPoint2[21310] = {X 486.2773, Y 8.1234, Z -3.0000, A 0.000, B 0.000, C 0.000 }
gfCNCPoint2[21311] = {X 486.9700, Y 8.1112, Z -3.0000, A 0.000, B 0.000, C 0.000 }
gfCNCPoint2[21312] = {X 492.3825, Y 8.1112, Z -3.0000, A 0.000, B 0.000, C 0.000 }
gfCNCPoint2[21313] = {X 492.3825, Y 4.1112, Z -3.0000, A 0.000, B 0.000, C 0.000 }
gfCNCPoint2[21314] = {X 492.3825, Y 8.1912, Z -3.0000, A 0.000, B 0.000, C 0.000 }
gfCNCPoint2[21315] = {X 502.2053, Y 8.1912, Z -3.0000, A 0.000, B 0.000, C 0.000 }
gfCNCPoint2[21316] = {X 502.7349, Y 8.1954, Z -3.0000, A 0.000, B 0.000, C 0.000 }
gfCNCPoint2[21317] = {X 503.6164, Y 8.3012, Z -3.0000, A 0.000, B 0.000, C 0.000 }
gfCNCPoint2[21318] = {X 504.4527, Y 8.5996, Z -3.0000, A 0.000, B 0.000, C 0.000 }
gfCNCPoint2[21319] = {X 505.2021, Y 9.0757, Z -3.0000, A 0.000, B 0.000, C 0.000 }
gfCNCPoint2[21320] = {X 505.8274, Y 9.7060, Z -3.0000, A 0.000, B 0.000, C 0.000 }
gfCNCPoint2[21321] = {X 506.2977, Y 10.4591, Z -3.0000, A 0.000, B 0.000, C 0.000 }
gfCNCPoint2[21322] = {X 506.5896, Y 11.2976, Z -3.0000, A 0.000, B 0.000, C 0.000 }
gfCNCPoint2[21323] = {X 506.6885, Y 12.1800, Z -3.0000, A 0.000, B 0.000, C 0.000 }
gfCNCPoint2[21324] = {X 506.6883, Y 13.0192, Z -3.0000, A 0.000, B 0.000, C 0.000 }
gfCNCPoint2[21325] = {X 506.5796, Y 13.9050, Z -3.0000, A 0.000, B 0.000, C 0.000 }
gfCNCPoint2[21326] = {X 506.2773, Y 14.7446, Z -3.0000, A 0.000, B 0.000, C 0.000 }
gfCNCPoint2[21327] = {X 505.7963, Y 15.4963, Z -3.0000, A 0.000, B 0.000, C 0.000 }
gfCNCPoint2[21328] = {X 505.1606, Y 16.1227, Z -3.0000, A 0.000, B 0.000, C 0.000 }
gfCNCPoint2[21329] = {X 505.1605, Y 41.0657, Z -3.0000, A 0.000, B 0.000, C 0.000 }
gfCNCPoint2[21330] = {X 505.2994, Y 41.1784, Z -3.0000, A 0.000, B 0.000, C 0.000 }
gfCNCPoint2[21331] = {X 505.8856, Y 41.8050, Z -3.0000, A 0.000, B 0.000, C 0.000 }
gfCNCPoint2[21332] = {X 506.3247, Y 42.5421, Z -3.0000, A 0.000, B 0.000, C 0.000 }
gfCNCPoint2[21333] = {X 506.5965, Y 43.3559, Z -3.0000, A 0.000, B 0.000, C 0.000 }
gfCNCPoint2[21334] = {X 506.6885, Y 44.2089, Z -3.0000, A 0.000, B 0.000, C 0.000 }
gfCNCPoint2[21335] = {X 506.6885, Y 45.0000, Z -3.0000, A 0.000, B 0.000, C 0.000 }
gfCNCPoint2[21336] = {X 506.5882, Y 45.8901, Z -3.0000, A 0.000, B 0.000, C 0.000 }
gfCNCPoint2[21337] = {X 506.2924, Y 46.7355, Z -3.0000, A 0.000, B 0.000, C 0.000 }
gfCNCPoint2[21338] = {X 505.8158, Y 47.4940, Z -3.0000, A 0.000, B 0.000, C 0.000 }
gfCNCPoint2[21339] = {X 505.1825, Y 48.1273, Z -3.0000, A 0.000, B 0.000, C 0.000 }
gfCNCPoint2[21340] = {X 504.4240, Y 48.6039, Z -3.0000, A 0.000, B 0.000, C 0.000 }
gfCNCPoint2[21341] = {X 503.5786, Y 48.8997, Z -3.0000, A 0.000, B 0.000, C 0.000 }
gfCNCPoint2[21342] = {X 502.6885, Y 49.0000, Z -3.0000, A 0.000, B 0.000, C 0.000 }
gfCNCPoint2[21343] = {X 496.2450, Y 49.0000, Z -3.0000, A 0.000, B 0.000, C 0.000 }
gfCNCPoint2[21344] = {X 495.3549, Y 48.8997, Z -3.0000, A 0.000, B 0.000, C 0.000 }
gfCNCPoint2[21345] = {X 494.5095, Y 48.6039, Z -3.0000, A 0.000, B 0.000, C 0.000 }
gfCNCPoint2[21346] = {X 493.7511, Y 48.1273, Z -3.0000, A 0.000, B 0.000, C 0.000 }
gfCNCPoint2[21347] = {X 493.1177, Y 47.4939, Z -3.0000, A 0.000, B 0.000, C 0.000 }
gfCNCPoint2[21348] = {X 492.6411, Y 46.7355, Z -3.0000, A 0.000, B 0.000, C 0.000 }
gfCNCPoint2[21349] = {X 492.3453, Y 45.8900, Z -3.0000, A 0.000, B 0.000, C 0.000 }
gfCNCPoint2[21350] = {X 492.2450, Y 45.0000, Z -3.0000, A 0.000, B 0.000, C 0.000 }
gfCNCPoint2[21351] = {X 492.2454, Y 44.1538, Z -3.0000, A 0.000, B 0.000, C 0.000 }
gfCNCPoint2[21352] = {X 492.3560, Y 43.2730, Z -3.0000, A 0.000, B 0.000, C 0.000 }
gfCNCPoint2[21353] = {X 492.6582, Y 42.4382, Z -3.0000, A 0.000, B 0.000, C 0.000 }
gfCNCPoint2[21354] = {X 493.1371, Y 41.6907, Z -3.0000, A 0.000, B 0.000, C 0.000 }
gfCNCPoint2[21355] = {X 493.7690, Y 41.0672, Z -3.0000, A 0.000, B 0.000, C 0.000 }
gfCNCPoint2[21356] = {X 493.7690, Y 34.1538, Z -3.0000, A 0.000, B 0.000, C 0.000 }
gfCNCPoint2[21357] = {X 490.7727, Y 34.1538, Z -3.0000, A 0.000, B 0.000, C 0.000 }
gfCNCPoint2[21358] = {X 490.5299, Y 34.1510, Z -3.0000, A 0.000, B 0.000, C 0.000 }
gfCNCPoint2[21359] = {X 486.0901, Y 42.7965, Z -3.0000, A 0.000, B 0.000, C 0.000 }
gfCNCPoint2[21360] = {X 486.1471, Y 42.9480, Z -3.0000, A 0.000, B 0.000, C 0.000 }
gfCNCPoint2[21361] = {X 486.2997, Y 43.5703, Z -3.0000, A 0.000, B 0.000, C 0.000 }
gfCNCPoint2[21362] = {X 486.3510, Y 44.2089, Z -3.0000, A 0.000, B 0.000, C 0.000 }
gfCNCPoint2[21363] = {X 486.3510, Y 45.0000, Z -3.0000, A 0.000, B 0.000, C 0.000 }
gfCNCPoint2[21364] = {X 486.2507, Y 45.8901, Z -3.0000, A 0.000, B 0.000, C 0.000 }
gfCNCPoint2[21365] = {X 485.9549, Y 46.7355, Z -3.0000, A 0.000, B 0.000, C 0.000 }
gfCNCPoint2[21366] = {X 485.4783, Y 47.4940, Z -3.0000, A 0.000, B 0.000, C 0.000 }
gfCNCPoint2[21367] = {X 484.8450, Y 48.1273, Z -3.0000, A 0.000, B 0.000, C 0.000 }
gfCNCPoint2[21368] = {X 484.0866, Y 48.6039, Z -3.0000, A 0.000, B 0.000, C 0.000 }
gfCNCPoint2[21369] = {X 483.2411, Y 48.8997, Z -3.0000, A 0.000, B 0.000, C 0.000 }
gfCNCPoint2[21370] = {X 482.3510, Y 49.0000, Z -3.0000, A 0.000, B 0.000, C 0.000 }
gfCNCPoint2[21371] = {X 475.7650, Y 49.0000, Z -3.0000, A 0.000, B 0.000, C 0.000 }
gfCNCPoint2[21372] = {X 474.8749, Y 48.8997, Z -3.0000, A 0.000, B 0.000, C 0.000 }
gfCNCPoint2[21373] = {X 474.0294, Y 48.6039, Z -3.0000, A 0.000, B 0.000, C 0.000 }
gfCNCPoint2[21374] = {X 473.2710, Y 48.1273, Z -3.0000, A 0.000, B 0.000, C 0.000 }
gfCNCPoint2[21375] = {X 472.6376, Y 47.4940, Z -3.0000, A 0.000, B 0.000, C 0.000 }
gfCNCPoint2[21376] = {X 472.1611, Y 46.7355, Z -3.0000, A 0.000, B 0.000, C 0.000 }
gfCNCPoint2[21377] = {X 471.8652, Y 45.8901, Z -3.0000, A 0.000, B 0.000, C 0.000 }
gfCNCPoint2[21378] = {X 471.7650, Y 45.0000, Z -3.0000, A 0.000, B 0.000, C 0.000 }
gfCNCPoint2[21379] = {X 471.7653, Y 44.1538, Z -3.0000, A 0.000, B 0.000, C 0.000 }
gfCNCPoint2[21380] = {X 471.8601, Y 43.3414, Z -3.0000, A 0.000, B 0.000, C 0.000 }
gfCNCPoint2[21381] = {X 472.1182, Y 42.5654, Z -3.0000, A 0.000, B 0.000, C 0.000 }
gfCNCPoint2[21382] = {X 472.5286, Y 41.8580, Z -3.0000, A 0.000, B 0.000, C 0.000 }
gfCNCPoint2[21383] = {X 473.0744, Y 41.2489, Z -3.0000, A 0.000, B 0.000, C 0.000 }
gfCNCPoint2[21384] = {X 473.7327, Y 40.7635, Z -3.0000, A 0.000, B 0.000, C 0.000 }
gfCNCPoint2[21385] = {X 474.4759, Y 40.4222, Z -3.0000, A 0.000, B 0.000, C 0.000 }
gfCNCPoint2[21386] = {X 478.6566, Y 32.2388, Z -3.0000, A 0.000, B 0.000, C 0.000 }
gfCNCPoint2[21387] = {X 477.3662, Y 31.3986, Z -3.0000, A 0.000, B 0.000, C 0.000 }
gfCNCPoint2[21388] = {X 476.2038, Y 30.3886, Z -3.0000, A 0.000, B 0.000, C 0.000 }
gfCNCPoint2[21389] = {X 475.1917, Y 29.2281, Z -3.0000, A 0.000, B 0.000, C 0.000 }
gfCNCPoint2[21390] = {X 474.3491, Y 27.9392, Z -3.0000, A 0.000, B 0.000, C 0.000 }
gfCNCPoint2[21391] = {X 473.6922, Y 26.5465, Z -3.0000, A 0.000, B 0.000, C 0.000 }
gfCNCPoint2[21392] = {X 473.2333, Y 25.0766, Z -3.0000, A 0.000, B 0.000, C 0.000 }
gfCNCPoint2[21393] = {X 472.9256, Y 23.4256, Z -3.0000, A 0.000, B 0.000, C 0.000 }
gfCNCPoint2[21394] = {X 472.7880, Y 21.7518, Z -3.0000, A 0.000, B 0.000, C 0.000 }
gfCNCPoint2[21395] = {X 472.8221, Y 20.0727, Z -3.0000, A 0.000, B 0.000, C 0.000 }
gfCNCPoint2[21396] = {X 473.0273, Y 18.4059, Z -3.0000, A 0.000, B 0.000, C 0.000 }
gfCNCPoint2[21397] = {X 473.4017, Y 16.7687, Z -3.0000, A 0.000, B 0.000, C 0.000 }
gfCNCPoint2[21398] = {X 473.9296, Y 15.2949, Z -3.0000, A 0.000, B 0.000, C 0.000 }
gfCNCPoint2[21399] = {X 474.6527, Y 13.9063, Z -3.0000, A 0.000, B 0.000, C 0.000 }
gfCNCPoint2[21400] = {X 475.5575, Y 12.6288, Z -3.0000, A 0.000, B 0.000, C 0.000 }
gfCNCPoint2[21401] = {X 476.6274, Y 11.4858, Z -3.0000, A 0.000, B 0.000, C 0.000 }
gfCNCPoint2[21402] = {X 477.8425, Y 10.4986, Z -3.0000, A 0.000, B 0.000, C 0.000 }
gfCNCPoint2[21403] = {X 479.1803, Y 9.6855, Z -3.0000, A 0.000, B 0.000, C 0.000 }
gfCNCPoint2[21404] = {X 480.6161, Y 9.0615, Z -3.0000, A 0.000, B 0.000, C 0.000 }
gfCNCPoint2[21405] = {X 482.1233, Y 8.6381, Z -3.0000, A 0.000, B 0.000, C 0.000 }
gfCNCPoint2[21406] = {X 484.1898, Y 8.3160, Z -3.0000, A 0.000, B 0.000, C 0.000 }
gfCNCPoint2[21407] = {X 486.2782, Y 8.2034, Z -3.0000, A 0.000, B 0.000, C 0.000 }
gfCNCPoint2[21408] = {X 486.9707, Y 8.1912, Z -3.0000, A 0.000, B 0.000, C 0.000 }
gfCNCPoint2[21409] = {X 492.3825, Y 8.1912, Z -3.0000, A 0.000, B 0.000, C 0.000 }
gfCNCPoint2[21410] = {X 492.3825, Y 4.1112, Z -3.0000, A 0.000, B 0.000, C 0.000 }
gfCNCPoint2[21411] = {X 492.3825, Y 4.1112, Z 0.0000, A 0.000, B 0.000, C 0.000 }
gfCNCPoint2[21412] = {X 492.3825, Y 4.1112, Z 11.0000, A 0.000, B 0.000, C 0.000 }
gfCNCPoint2[21413] = {X 533.9640, Y 3.7910, Z 11.0000, A 0.000, B 0.000, C 0.000 }
gfCNCPoint2[21414] = {X 533.9640, Y 3.7910, Z 0.0000, A 0.000, B 0.000, C 0.000 }
gfCNCPoint2[21415] = {X 533.9640, Y 3.7910, Z -3.0000, A 0.000, B 0.000, C 0.000 }
gfCNCPoint2[21416] = {X 533.9639, Y 7.8710, Z -3.0000, A 0.000, B 0.000, C 0.000 }
gfCNCPoint2[21417] = {X 543.7499, Y 7.8712, Z -3.0000, A 0.000, B 0.000, C 0.000 }
gfCNCPoint2[21418] = {X 544.7300, Y 7.9568, Z -3.0000, A 0.000, B 0.000, C 0.000 }
gfCNCPoint2[21419] = {X 545.6655, Y 8.2616, Z -3.0000, A 0.000, B 0.000, C 0.000 }
gfCNCPoint2[21420] = {X 546.5078, Y 8.7699, Z -3.0000, A 0.000, B 0.000, C 0.000 }
gfCNCPoint2[21421] = {X 547.2135, Y 9.4555, Z -3.0000, A 0.000, B 0.000, C 0.000 }
gfCNCPoint2[21422] = {X 547.7459, Y 10.2828, Z -3.0000, A 0.000, B 0.000, C 0.000 }
gfCNCPoint2[21423] = {X 548.0776, Y 11.2090, Z -3.0000, A 0.000, B 0.000, C 0.000 }
gfCNCPoint2[21424] = {X 548.1914, Y 12.1863, Z -3.0000, A 0.000, B 0.000, C 0.000 }
gfCNCPoint2[21425] = {X 548.1912, Y 13.0225, Z -3.0000, A 0.000, B 0.000, C 0.000 }
gfCNCPoint2[21426] = {X 548.0827, Y 13.9407, Z -3.0000, A 0.000, B 0.000, C 0.000 }
gfCNCPoint2[21427] = {X 547.7813, Y 14.8148, Z -3.0000, A 0.000, B 0.000, C 0.000 }
gfCNCPoint2[21428] = {X 547.3008, Y 15.6047, Z -3.0000, A 0.000, B 0.000, C 0.000 }
gfCNCPoint2[21429] = {X 546.6632, Y 16.2743, Z -3.0000, A 0.000, B 0.000, C 0.000 }
gfCNCPoint2[21430] = {X 546.6634, Y 40.9133, Z -3.0000, A 0.000, B 0.000, C 0.000 }
gfCNCPoint2[21431] = {X 546.6857, Y 40.9312, Z -3.0000, A 0.000, B 0.000, C 0.000 }
gfCNCPoint2[21432] = {X 547.3157, Y 41.6012, Z -3.0000, A 0.000, B 0.000, C 0.000 }
gfCNCPoint2[21433] = {X 547.7895, Y 42.3892, Z -3.0000, A 0.000, B 0.000, C 0.000 }
gfCNCPoint2[21434] = {X 548.0859, Y 43.2598, Z -3.0000, A 0.000, B 0.000, C 0.000 }
gfCNCPoint2[21435] = {X 548.1913, Y 44.1733, Z -3.0000, A 0.000, B 0.000, C 0.000 }
gfCNCPoint2[21436] = {X 548.1914, Y 45.0006, Z -3.0000, A 0.000, B 0.000, C 0.000 }
gfCNCPoint2[21437] = {X 548.0776, Y 45.9778, Z -3.0000, A 0.000, B 0.000, C 0.000 }
gfCNCPoint2[21438] = {X 547.7459, Y 46.9040, Z -3.0000, A 0.000, B 0.000, C 0.000 }
gfCNCPoint2[21439] = {X 547.2135, Y 47.7313, Z -3.0000, A 0.000, B 0.000, C 0.000 }
gfCNCPoint2[21440] = {X 546.5078, Y 48.4168, Z -3.0000, A 0.000, B 0.000, C 0.000 }
gfCNCPoint2[21441] = {X 545.6654, Y 48.9251, Z -3.0000, A 0.000, B 0.000, C 0.000 }
gfCNCPoint2[21442] = {X 544.7300, Y 49.2298, Z -3.0000, A 0.000, B 0.000, C 0.000 }
gfCNCPoint2[21443] = {X 543.7499, Y 49.3153, Z -3.0000, A 0.000, B 0.000, C 0.000 }
gfCNCPoint2[21444] = {X 524.0449, Y 49.3158, Z -3.0000, A 0.000, B 0.000, C 0.000 }
gfCNCPoint2[21445] = {X 523.4983, Y 49.9497, Z -3.0000, A 0.000, B 0.000, C 0.000 }
gfCNCPoint2[21446] = {X 522.8434, Y 50.4709, Z -3.0000, A 0.000, B 0.000, C 0.000 }
gfCNCPoint2[21447] = {X 522.1029, Y 50.8611, Z -3.0000, A 0.000, B 0.000, C 0.000 }
gfCNCPoint2[21448] = {X 521.3028, Y 51.1067, Z -3.0000, A 0.000, B 0.000, C 0.000 }
gfCNCPoint2[21449] = {X 520.4709, Y 51.1991, Z -3.0000, A 0.000, B 0.000, C 0.000 }
gfCNCPoint2[21450] = {X 519.7998, Y 51.1991, Z -3.0000, A 0.000, B 0.000, C 0.000 }
gfCNCPoint2[21451] = {X 518.8385, Y 51.0908, Z -3.0000, A 0.000, B 0.000, C 0.000 }
gfCNCPoint2[21452] = {X 517.9254, Y 50.7713, Z -3.0000, A 0.000, B 0.000, C 0.000 }
gfCNCPoint2[21453] = {X 517.1063, Y 50.2566, Z -3.0000, A 0.000, B 0.000, C 0.000 }
gfCNCPoint2[21454] = {X 516.4223, Y 49.5726, Z -3.0000, A 0.000, B 0.000, C 0.000 }
gfCNCPoint2[21455] = {X 515.9076, Y 48.7535, Z -3.0000, A 0.000, B 0.000, C 0.000 }
gfCNCPoint2[21456] = {X 515.5881, Y 47.8404, Z -3.0000, A 0.000, B 0.000, C 0.000 }
gfCNCPoint2[21457] = {X 515.4798, Y 46.8791, Z -3.0000, A 0.000, B 0.000, C 0.000 }
gfCNCPoint2[21458] = {X 515.4798, Y 39.9011, Z -3.0000, A 0.000, B 0.000, C 0.000 }
gfCNCPoint2[21459] = {X 515.5869, Y 38.9451, Z -3.0000, A 0.000, B 0.000, C 0.000 }
gfCNCPoint2[21460] = {X 515.9029, Y 38.0365, Z -3.0000, A 0.000, B 0.000, C 0.000 }
gfCNCPoint2[21461] = {X 516.4121, Y 37.2204, Z -3.0000, A 0.000, B 0.000, C 0.000 }
gfCNCPoint2[21462] = {X 517.0893, Y 36.5372, Z -3.0000, A 0.000, B 0.000, C 0.000 }
gfCNCPoint2[21463] = {X 517.9010, Y 36.0208, Z -3.0000, A 0.000, B 0.000, C 0.000 }
gfCNCPoint2[21464] = {X 518.8067, Y 35.6968, Z -3.0000, A 0.000, B 0.000, C 0.000 }
gfCNCPoint2[21465] = {X 519.7617, Y 35.5813, Z -3.0000, A 0.000, B 0.000, C 0.000 }
gfCNCPoint2[21466] = {X 520.5269, Y 35.5815, Z -3.0000, A 0.000, B 0.000, C 0.000 }
gfCNCPoint2[21467] = {X 521.3535, Y 35.6728, Z -3.0000, A 0.000, B 0.000, C 0.000 }
gfCNCPoint2[21468] = {X 522.1473, Y 35.9208, Z -3.0000, A 0.000, B 0.000, C 0.000 }
gfCNCPoint2[21469] = {X 522.8788, Y 36.3163, Z -3.0000, A 0.000, B 0.000, C 0.000 }
gfCNCPoint2[21470] = {X 523.5211, Y 36.8446, Z -3.0000, A 0.000, B 0.000, C 0.000 }
gfCNCPoint2[21471] = {X 524.0502, Y 37.4862, Z -3.0000, A 0.000, B 0.000, C 0.000 }
gfCNCPoint2[21472] = {X 534.6319, Y 37.4867, Z -3.0000, A 0.000, B 0.000, C 0.000 }
gfCNCPoint2[21473] = {X 534.6319, Y 33.9650, Z -3.0000, A 0.000, B 0.000, C 0.000 }
gfCNCPoint2[21474] = {X 530.1091, Y 33.9663, Z -3.0000, A 0.000, B 0.000, C 0.000 }
gfCNCPoint2[21475] = {X 529.5769, Y 34.6104, Z -3.0000, A 0.000, B 0.000, C 0.000 }
gfCNCPoint2[21476] = {X 528.9307, Y 35.1399, Z -3.0000, A 0.000, B 0.000, C 0.000 }
gfCNCPoint2[21477] = {X 528.1946, Y 35.5352, Z -3.0000, A 0.000, B 0.000, C 0.000 }
gfCNCPoint2[21478] = {X 527.3963, Y 35.7814, Z -3.0000, A 0.000, B 0.000, C 0.000 }
gfCNCPoint2[21479] = {X 526.5655, Y 35.8693, Z -3.0000, A 0.000, B 0.000, C 0.000 }
gfCNCPoint2[21480] = {X 525.8868, Y 35.8694, Z -3.0000, A 0.000, B 0.000, C 0.000 }
gfCNCPoint2[21481] = {X 524.9255, Y 35.7611, Z -3.0000, A 0.000, B 0.000, C 0.000 }
gfCNCPoint2[21482] = {X 524.0124, Y 35.4416, Z -3.0000, A 0.000, B 0.000, C 0.000 }
gfCNCPoint2[21483] = {X 523.1933, Y 34.9270, Z -3.0000, A 0.000, B 0.000, C 0.000 }
gfCNCPoint2[21484] = {X 522.5092, Y 34.2429, Z -3.0000, A 0.000, B 0.000, C 0.000 }
gfCNCPoint2[21485] = {X 521.9946, Y 33.4238, Z -3.0000, A 0.000, B 0.000, C 0.000 }
gfCNCPoint2[21486] = {X 521.6751, Y 32.5107, Z -3.0000, A 0.000, B 0.000, C 0.000 }
gfCNCPoint2[21487] = {X 521.5668, Y 31.5495, Z -3.0000, A 0.000, B 0.000, C 0.000 }
gfCNCPoint2[21488] = {X 521.5668, Y 24.5714, Z -3.0000, A 0.000, B 0.000, C 0.000 }
gfCNCPoint2[21489] = {X 521.6739, Y 23.6153, Z -3.0000, A 0.000, B 0.000, C 0.000 }
gfCNCPoint2[21490] = {X 521.9900, Y 22.7066, Z -3.0000, A 0.000, B 0.000, C 0.000 }
gfCNCPoint2[21491] = {X 522.4994, Y 21.8904, Z -3.0000, A 0.000, B 0.000, C 0.000 }
gfCNCPoint2[21492] = {X 523.1768, Y 21.2071, Z -3.0000, A 0.000, B 0.000, C 0.000 }
gfCNCPoint2[21493] = {X 523.9886, Y 20.6908, Z -3.0000, A 0.000, B 0.000, C 0.000 }
gfCNCPoint2[21494] = {X 524.8946, Y 20.3669, Z -3.0000, A 0.000, B 0.000, C 0.000 }
gfCNCPoint2[21495] = {X 525.8498, Y 20.2516, Z -3.0000, A 0.000, B 0.000, C 0.000 }
gfCNCPoint2[21496] = {X 526.5695, Y 20.2516, Z -3.0000, A 0.000, B 0.000, C 0.000 }
gfCNCPoint2[21497] = {X 527.3947, Y 20.3392, Z -3.0000, A 0.000, B 0.000, C 0.000 }
gfCNCPoint2[21498] = {X 528.1879, Y 20.5829, Z -3.0000, A 0.000, B 0.000, C 0.000 }
gfCNCPoint2[21499] = {X 528.9199, Y 20.9737, Z -3.0000, A 0.000, B 0.000, C 0.000 }
gfCNCPoint2[21500] = {X 529.5636, Y 21.4974, Z -3.0000, A 0.000, B 0.000, C 0.000 }
gfCNCPoint2[21501] = {X 530.0954, Y 22.1344, Z -3.0000, A 0.000, B 0.000, C 0.000 }
gfCNCPoint2[21502] = {X 534.6319, Y 22.1347, Z -3.0000, A 0.000, B 0.000, C 0.000 }
gfCNCPoint2[21503] = {X 534.6319, Y 19.7014, Z -3.0000, A 0.000, B 0.000, C 0.000 }
gfCNCPoint2[21504] = {X 524.1925, Y 19.7010, Z -3.0000, A 0.000, B 0.000, C 0.000 }
gfCNCPoint2[21505] = {X 523.6601, Y 20.3458, Z -3.0000, A 0.000, B 0.000, C 0.000 }
gfCNCPoint2[21506] = {X 523.0134, Y 20.8760, Z -3.0000, A 0.000, B 0.000, C 0.000 }
gfCNCPoint2[21507] = {X 522.2767, Y 21.2716, Z -3.0000, A 0.000, B 0.000, C 0.000 }
gfCNCPoint2[21508] = {X 521.4776, Y 21.5179, Z -3.0000, A 0.000, B 0.000, C 0.000 }
gfCNCPoint2[21509] = {X 520.6460, Y 21.6056, Z -3.0000, A 0.000, B 0.000, C 0.000 }
gfCNCPoint2[21510] = {X 519.9691, Y 21.6057, Z -3.0000, A 0.000, B 0.000, C 0.000 }
gfCNCPoint2[21511] = {X 519.0078, Y 21.4974, Z -3.0000, A 0.000, B 0.000, C 0.000 }
gfCNCPoint2[21512] = {X 518.0947, Y 21.1779, Z -3.0000, A 0.000, B 0.000, C 0.000 }
gfCNCPoint2[21513] = {X 517.2756, Y 20.6632, Z -3.0000, A 0.000, B 0.000, C 0.000 }
gfCNCPoint2[21514] = {X 516.5916, Y 19.9792, Z -3.0000, A 0.000, B 0.000, C 0.000 }
gfCNCPoint2[21515] = {X 516.0769, Y 19.1601, Z -3.0000, A 0.000, B 0.000, C 0.000 }
gfCNCPoint2[21516] = {X 515.7574, Y 18.2470, Z -3.0000, A 0.000, B 0.000, C 0.000 }
gfCNCPoint2[21517] = {X 515.6491, Y 17.2857, Z -3.0000, A 0.000, B 0.000, C 0.000 }
gfCNCPoint2[21518] = {X 515.6491, Y 10.3077, Z -3.0000, A 0.000, B 0.000, C 0.000 }
gfCNCPoint2[21519] = {X 515.7562, Y 9.3519, Z -3.0000, A 0.000, B 0.000, C 0.000 }
gfCNCPoint2[21520] = {X 516.0720, Y 8.4435, Z -3.0000, A 0.000, B 0.000, C 0.000 }
gfCNCPoint2[21521] = {X 516.5811, Y 7.6275, Z -3.0000, A 0.000, B 0.000, C 0.000 }
gfCNCPoint2[21522] = {X 517.2580, Y 6.9443, Z -3.0000, A 0.000, B 0.000, C 0.000 }
gfCNCPoint2[21523] = {X 518.0693, Y 6.4278, Z -3.0000, A 0.000, B 0.000, C 0.000 }
gfCNCPoint2[21524] = {X 518.9748, Y 6.1037, Z -3.0000, A 0.000, B 0.000, C 0.000 }
gfCNCPoint2[21525] = {X 519.9296, Y 5.9879, Z -3.0000, A 0.000, B 0.000, C 0.000 }
gfCNCPoint2[21526] = {X 520.6502, Y 5.9879, Z -3.0000, A 0.000, B 0.000, C 0.000 }
gfCNCPoint2[21527] = {X 521.4757, Y 6.0752, Z -3.0000, A 0.000, B 0.000, C 0.000 }
gfCNCPoint2[21528] = {X 522.2693, Y 6.3188, Z -3.0000, A 0.000, B 0.000, C 0.000 }
gfCNCPoint2[21529] = {X 523.0017, Y 6.7097, Z -3.0000, A 0.000, B 0.000, C 0.000 }
gfCNCPoint2[21530] = {X 523.6458, Y 7.2334, Z -3.0000, A 0.000, B 0.000, C 0.000 }
gfCNCPoint2[21531] = {X 524.1778, Y 7.8707, Z -3.0000, A 0.000, B 0.000, C 0.000 }
gfCNCPoint2[21532] = {X 533.9639, Y 7.8710, Z -3.0000, A 0.000, B 0.000, C 0.000 }
gfCNCPoint2[21533] = {X 533.9640, Y 3.8710, Z -3.0000, A 0.000, B 0.000, C 0.000 }
gfCNCPoint2[21534] = {X 533.9639, Y 7.9510, Z -3.0000, A 0.000, B 0.000, C 0.000 }
gfCNCPoint2[21535] = {X 543.7510, Y 7.9512, Z -3.0000, A 0.000, B 0.000, C 0.000 }
gfCNCPoint2[21536] = {X 544.7132, Y 8.0350, Z -3.0000, A 0.000, B 0.000, C 0.000 }
gfCNCPoint2[21537] = {X 545.6315, Y 8.3340, Z -3.0000, A 0.000, B 0.000, C 0.000 }
gfCNCPoint2[21538] = {X 546.4585, Y 8.8329, Z -3.0000, A 0.000, B 0.000, C 0.000 }
gfCNCPoint2[21539] = {X 547.1513, Y 9.5058, Z -3.0000, A 0.000, B 0.000, C 0.000 }
gfCNCPoint2[21540] = {X 547.6740, Y 10.3179, Z -3.0000, A 0.000, B 0.000, C 0.000 }
gfCNCPoint2[21541] = {X 547.9997, Y 11.2271, Z -3.0000, A 0.000, B 0.000, C 0.000 }
gfCNCPoint2[21542] = {X 548.1114, Y 12.1864, Z -3.0000, A 0.000, B 0.000, C 0.000 }
gfCNCPoint2[21543] = {X 548.1112, Y 13.0217, Z -3.0000, A 0.000, B 0.000, C 0.000 }
gfCNCPoint2[21544] = {X 548.0026, Y 13.9319, Z -3.0000, A 0.000, B 0.000, C 0.000 }
gfCNCPoint2[21545] = {X 547.7010, Y 14.7975, Z -3.0000, A 0.000, B 0.000, C 0.000 }
gfCNCPoint2[21546] = {X 547.2204, Y 15.5780, Z -3.0000, A 0.000, B 0.000, C 0.000 }
gfCNCPoint2[21547] = {X 546.5832, Y 16.2370, Z -3.0000, A 0.000, B 0.000, C 0.000 }
gfCNCPoint2[21548] = {X 546.5834, Y 40.9515, Z -3.0000, A 0.000, B 0.000, C 0.000 }
gfCNCPoint2[21549] = {X 546.6345, Y 40.9927, Z -3.0000, A 0.000, B 0.000, C 0.000 }
gfCNCPoint2[21550] = {X 547.2524, Y 41.6502, Z -3.0000, A 0.000, B 0.000, C 0.000 }
gfCNCPoint2[21551] = {X 547.7172, Y 42.4235, Z -3.0000, A 0.000, B 0.000, C 0.000 }
gfCNCPoint2[21552] = {X 548.0079, Y 43.2776, Z -3.0000, A 0.000, B 0.000, C 0.000 }
gfCNCPoint2[21553] = {X 548.1113, Y 44.1740, Z -3.0000, A 0.000, B 0.000, C 0.000 }
gfCNCPoint2[21554] = {X 548.1114, Y 45.0004, Z -3.0000, A 0.000, B 0.000, C 0.000 }
gfCNCPoint2[21555] = {X 547.9997, Y 45.9597, Z -3.0000, A 0.000, B 0.000, C 0.000 }
gfCNCPoint2[21556] = {X 547.6740, Y 46.8689, Z -3.0000, A 0.000, B 0.000, C 0.000 }
gfCNCPoint2[21557] = {X 547.1513, Y 47.6810, Z -3.0000, A 0.000, B 0.000, C 0.000 }
gfCNCPoint2[21558] = {X 546.4585, Y 48.3538, Z -3.0000, A 0.000, B 0.000, C 0.000 }
gfCNCPoint2[21559] = {X 545.6315, Y 48.8526, Z -3.0000, A 0.000, B 0.000, C 0.000 }
gfCNCPoint2[21560] = {X 544.7131, Y 49.1516, Z -3.0000, A 0.000, B 0.000, C 0.000 }
gfCNCPoint2[21561] = {X 543.7510, Y 49.2353, Z -3.0000, A 0.000, B 0.000, C 0.000 }
gfCNCPoint2[21562] = {X 524.0033, Y 49.2358, Z -3.0000, A 0.000, B 0.000, C 0.000 }
gfCNCPoint2[21563] = {X 523.4666, Y 49.8690, Z -3.0000, A 0.000, B 0.000, C 0.000 }
gfCNCPoint2[21564] = {X 522.8205, Y 50.3902, Z -3.0000, A 0.000, B 0.000, C 0.000 }
gfCNCPoint2[21565] = {X 522.0880, Y 50.7807, Z -3.0000, A 0.000, B 0.000, C 0.000 }
gfCNCPoint2[21566] = {X 521.2951, Y 51.0266, Z -3.0000, A 0.000, B 0.000, C 0.000 }
gfCNCPoint2[21567] = {X 520.4702, Y 51.1191, Z -3.0000, A 0.000, B 0.000, C 0.000 }
gfCNCPoint2[21568] = {X 519.7998, Y 51.1191, Z -3.0000, A 0.000, B 0.000, C 0.000 }
gfCNCPoint2[21569] = {X 518.8563, Y 51.0128, Z -3.0000, A 0.000, B 0.000, C 0.000 }
gfCNCPoint2[21570] = {X 517.9601, Y 50.6992, Z -3.0000, A 0.000, B 0.000, C 0.000 }
gfCNCPoint2[21571] = {X 517.1562, Y 50.1941, Z -3.0000, A 0.000, B 0.000, C 0.000 }
gfCNCPoint2[21572] = {X 516.4848, Y 49.5227, Z -3.0000, A 0.000, B 0.000, C 0.000 }
gfCNCPoint2[21573] = {X 515.9797, Y 48.7188, Z -3.0000, A 0.000, B 0.000, C 0.000 }
gfCNCPoint2[21574] = {X 515.6661, Y 47.8226, Z -3.0000, A 0.000, B 0.000, C 0.000 }
gfCNCPoint2[21575] = {X 515.5598, Y 46.8791, Z -3.0000, A 0.000, B 0.000, C 0.000 }
gfCNCPoint2[21576] = {X 515.5598, Y 39.9011, Z -3.0000, A 0.000, B 0.000, C 0.000 }
gfCNCPoint2[21577] = {X 515.6649, Y 38.9628, Z -3.0000, A 0.000, B 0.000, C 0.000 }
gfCNCPoint2[21578] = {X 515.9751, Y 38.0710, Z -3.0000, A 0.000, B 0.000, C 0.000 }
gfCNCPoint2[21579] = {X 516.4749, Y 37.2700, Z -3.0000, A 0.000, B 0.000, C 0.000 }
gfCNCPoint2[21580] = {X 517.1395, Y 36.5995, Z -3.0000, A 0.000, B 0.000, C 0.000 }
gfCNCPoint2[21581] = {X 517.9361, Y 36.0926, Z -3.0000, A 0.000, B 0.000, C 0.000 }
gfCNCPoint2[21582] = {X 518.8251, Y 35.7746, Z -3.0000, A 0.000, B 0.000, C 0.000 }
gfCNCPoint2[21583] = {X 519.7624, Y 35.6613, Z -3.0000, A 0.000, B 0.000, C 0.000 }
gfCNCPoint2[21584] = {X 520.5258, Y 35.6615, Z -3.0000, A 0.000, B 0.000, C 0.000 }
gfCNCPoint2[21585] = {X 521.3454, Y 35.7528, Z -3.0000, A 0.000, B 0.000, C 0.000 }
gfCNCPoint2[21586] = {X 522.1318, Y 36.0011, Z -3.0000, A 0.000, B 0.000, C 0.000 }
gfCNCPoint2[21587] = {X 522.8553, Y 36.3969, Z -3.0000, A 0.000, B 0.000, C 0.000 }
gfCNCPoint2[21588] = {X 523.4884, Y 36.9253, Z -3.0000, A 0.000, B 0.000, C 0.000 }
gfCNCPoint2[21589] = {X 524.0074, Y 37.5662, Z -3.0000, A 0.000, B 0.000, C 0.000 }
gfCNCPoint2[21590] = {X 534.7119, Y 37.5667, Z -3.0000, A 0.000, B 0.000, C 0.000 }
gfCNCPoint2[21591] = {X 534.7119, Y 33.8850, Z -3.0000, A 0.000, B 0.000, C 0.000 }
gfCNCPoint2[21592] = {X 530.0659, Y 33.8845, Z -3.0000, A 0.000, B 0.000, C 0.000 }
gfCNCPoint2[21593] = {X 530.0420, Y 33.9227, Z -3.0000, A 0.000, B 0.000, C 0.000 }
gfCNCPoint2[21594] = {X 529.5197, Y 34.5545, Z -3.0000, A 0.000, B 0.000, C 0.000 }
gfCNCPoint2[21595] = {X 528.8855, Y 35.0739, Z -3.0000, A 0.000, B 0.000, C 0.000 }
gfCNCPoint2[21596] = {X 528.1633, Y 35.4616, Z -3.0000, A 0.000, B 0.000, C 0.000 }
gfCNCPoint2[21597] = {X 527.3799, Y 35.7031, Z -3.0000, A 0.000, B 0.000, C 0.000 }
gfCNCPoint2[21598] = {X 526.5648, Y 35.7893, Z -3.0000, A 0.000, B 0.000, C 0.000 }
gfCNCPoint2[21599] = {X 525.8868, Y 35.7894, Z -3.0000, A 0.000, B 0.000, C 0.000 }
gfCNCPoint2[21600] = {X 524.9433, Y 35.6831, Z -3.0000, A 0.000, B 0.000, C 0.000 }
gfCNCPoint2[21601] = {X 524.0471, Y 35.3696, Z -3.0000, A 0.000, B 0.000, C 0.000 }
gfCNCPoint2[21602] = {X 523.2432, Y 34.8644, Z -3.0000, A 0.000, B 0.000, C 0.000 }
